KUKA KRL program: EPS_2_25694_BR06_A_20251117072402.src

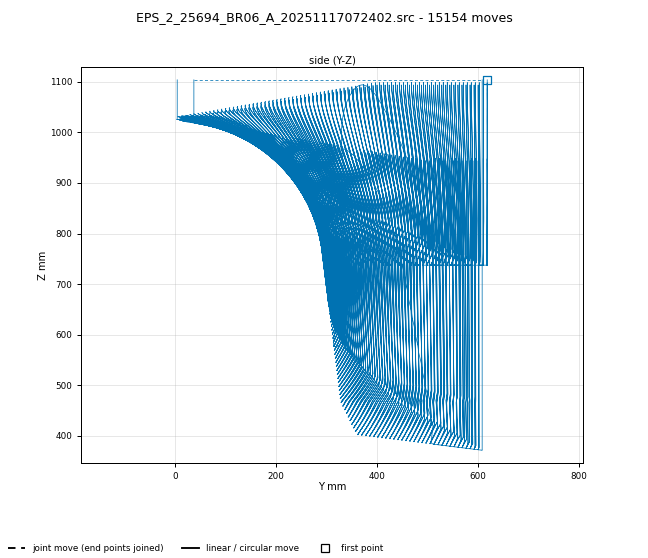
[picture p0: tool path of EPS_2_25694_BR06_A_20251117072402.src, 15154 of 15156 moves have a stored position in this frame; points joined in program order, loops and branches not executed]
&ACCESS RVP
&REL 4
&COMMENT QRS 19112012
&PARAM EDITMASK = *
DEF PART()
EXT BAS (BAS_COMMAND :IN,REAL :IN )
INT I
BAS (#INITMOV,0 )

;KUKA QRS Post kuka4.cps  Date:22-06-2017 !

File_ID=2908

QRS_PRE_INIT()

;Init var - Until changes are made in qrs_pre_init
Outlet_Square_prg=0
Inlet_1_Square_prg=0
Inlet_2_Square_prg=0
Inlet_3_Square_prg=0
Inlet_4_Square_prg=0
Inlet_5_Square_prg=0

Outlet_1={X 0.000, Y 400.000, Z 789.000, B 0.000, E1 0.000 }
Inlet_1={X 0.000, Y 466.000, Z 645.500, B 0.000, E1 180.000 }
Outlet_1_type=610
Inlet_1_type=457
;QRS#1=Sidecore dimensions
;QRS#2=600-24" Concrete
;QRS#3=450-18" Concrete
;QRS#4=
;QRS#5=
;QRS#6=
;QRS#7=
;QRS#8=
;QRS#9=S306-34L
;QRS#10=28A PSX-2
;QRS#11=
;QRS#12=
;QRS#13=
;QRS#14=
;QRS#15=
;QRS#16=1220x127x1448 4,75'
;QRS#17=EPS Height
;QRS#18=1094
;QRS#19=*
;QRS#20= UPDATED VERSION 22-06-2017
;QRS#21=*
Outlet_Square=0450
Inlet_1_Square=0250
Inlet_2_Square=0
Inlet_3_Square=0
Inlet_4_Square=0
Inlet_5_Square=0
Mill_Square=1
Outlet_Square_Prg=264
Inlet_1_Square_prg=274

QRS_INIT()

$ADVANCE=5

; T1
PTP {E1 171.024,E2 171.024}
PTP {X 0,Y 617.83,A -85,B 0,C 180,E1 171.024,E2 171.024,E3 0,E4 0,E5 0,E6 0}
QRS_SPEED_INIT()
LIN {X 0,Y 617.83,Z 1104,A -85,B 0,C 180,E1 171.024,E2 171.024,E3 0,E4 0,E5 0,E6 0} C_VEL
LIN {X 0,Y 617.83,Z 739.44,A -85,B 0,C 180,E1 171.024,E2 171.024} C_VEL
LIN {X 0,Y 617.865,Z 737.44,A -85,B 0,C 180,E1 171.21,E2 171.21} C_VEL
LIN {X 0,Y 618.044,Z 737.44,A -85,B 0,C 180,E1 171.886,E2 171.886} C_VEL
LIN {X 0,Y 618.018,Z 737.44,A -85,B 0,C 180,E1 176.532,E2 176.532} C_VEL
LIN {X 0,Y 618.01,Z 737.44,A -85,B 0,C 180,E1 181.155,E2 181.155} C_VEL
LIN {X 0,Y 617.998,Z 737.44,A -85,B 0,C 180,E1 185.786,E2 185.786} C_VEL
LIN {X 0,Y 618.001,Z 737.44,A -85,B 0,C 180,E1 190.456,E2 190.456} C_VEL
LIN {X 0,Y 617.923,Z 737.44,A -85,B 0,C 180,E1 195.199,E2 195.199} C_VEL
LIN {X 0,Y 617.894,Z 737.44,A -85,B 0,C 180,E1 200.05,E2 200.05} C_VEL
LIN {X 0,Y 617.438,Z 737.44,A -85,B 0,C 180,E1 202.548,E2 202.548} C_VEL
LIN {X 0,Y 617.919,Z 737.44,A -85,B 0,C 180,E1 205.056,E2 205.056} C_VEL
LIN {X 0,Y 617.398,Z 737.44,A -85,B 0,C 180,E1 207.66,E2 207.66} C_VEL
LIN {X 0,Y 617.828,Z 737.44,A -85,B 0,C 180,E1 210.281,E2 210.281} C_VEL
LIN {X 0,Y 617.3,Z 737.44,A -85,B 0,C 180,E1 213.028,E2 213.028} C_VEL
LIN {X 0,Y 617.772,Z 737.44,A -85,B 0,C 180,E1 215.801,E2 215.801} C_VEL
LIN {X 0,Y 617.531,Z 737.44,A -85,B 0,C 180,E1 218.094,E2 218.094} C_VEL
LIN {X 0,Y 617.504,Z 737.44,A -85,B 0,C 180,E1 218.725,E2 218.725} C_VEL
LIN {X 0,Y 617.717,Z 737.44,A -85,B 0,C 180,E1 221.737,E2 221.737} C_VEL
LIN {X 0,Y 617.832,Z 737.44,A -85,B 0,C 180,E1 225.095,E2 225.095} C_VEL
LIN {X 0,Y 617.441,Z 737.44,A -85,B 0,C 180,E1 228.309,E2 228.309} C_VEL
LIN {X 0,Y 617.823,Z 737.44,A -85,B 0,C 180,E1 231.298,E2 231.298} C_VEL
LIN {X 0,Y 617.894,Z 737.44,A -85,B 0,C 180,E1 235.778,E2 235.778} C_VEL
LIN {X 0,Y 617.659,Z 737.44,A -85,B 0,C 180,E1 236.368,E2 236.368} C_VEL
LIN {X 0,Y 616.896,Z 737.475,A -85,B 0,C 180,E1 236.468,E2 236.468} C_VEL
LIN {X 0,Y 617.501,Z 807.52,A -85,B 0,C 180,E1 237.463,E2 237.463} C_VEL
LIN {X 0,Y 617.519,Z 821.027,A -85,B 0,C 180,E1 237.687,E2 237.687} C_VEL
LIN {X 0,Y 617.637,Z 835.781,A -85,B 0,C 180,E1 238.01,E2 238.01} C_VEL
LIN {X 0,Y 617.583,Z 847.979,A -85,B 0,C 180,E1 238.328,E2 238.328} C_VEL
LIN {X 0,Y 617.775,Z 865.118,A -85,B 0,C 180,E1 238.871,E2 238.871} C_VEL
LIN {X 0,Y 617.661,Z 879.46,A -85,B 0,C 180,E1 239.394,E2 239.394} C_VEL
LIN {X 0,Y 617.795,Z 895.272,A -85,B 0,C 180,E1 240.077,E2 240.077} C_VEL
LIN {X 0,Y 617.796,Z 909.603,A -85,B 0,C 180,E1 240.772,E2 240.772} C_VEL
LIN {X 0,Y 617.753,Z 921.6,A -85,B 0,C 180,E1 241.411,E2 241.411} C_VEL
LIN {X 0,Y 617.843,Z 936.189,A -85,B 0,C 180,E1 242.286,E2 242.286} C_VEL
LIN {X 0,Y 617.842,Z 949.624,A -85,B 0,C 180,E1 243.174,E2 243.174} C_VEL
LIN {X 0,Y 617.833,Z 961.892,A -85,B 0,C 180,E1 244.06,E2 244.06} C_VEL
LIN {X 0,Y 617.824,Z 973.111,A -85,B 0,C 180,E1 244.94,E2 244.94} C_VEL
LIN {X 0,Y 617.855,Z 984.21,A -85,B 0,C 180,E1 245.886,E2 245.886} C_VEL
LIN {X 0,Y 617.904,Z 995.178,A -85,B 0,C 180,E1 246.901,E2 246.901} C_VEL
LIN {X 0,Y 617.833,Z 1005.53,A -85,B 0,C 180,E1 247.935,E2 247.935} C_VEL
LIN {X 0,Y 617.852,Z 1015.52,A -85,B 0,C 180,E1 249.023,E2 249.023} C_VEL
LIN {X 0,Y 617.958,Z 1024.894,A -85,B 0,C 180,E1 250.135,E2 250.135} C_VEL
LIN {X 0,Y 617.806,Z 1033.458,A -85,B 0,C 180,E1 251.226,E2 251.226} C_VEL
LIN {X 0,Y 617.799,Z 1041.796,A -85,B 0,C 180,E1 252.389,E2 252.389} C_VEL
LIN {X 0,Y 618,Z 1049.733,A -85,B 0,C 180,E1 253.612,E2 253.612} C_VEL
LIN {X 0,Y 617.809,Z 1056.882,A -85,B 0,C 180,E1 254.799,E2 254.799} C_VEL
LIN {X 0,Y 617.809,Z 1064.812,A -85,B 0,C 180,E1 256.29,E2 256.29} C_VEL
LIN {X 0,Y 617.96,Z 1070.477,A -85,B 0,C 180,E1 257.48,E2 257.48} C_VEL
LIN {X 0,Y 617.732,Z 1076.732,A -85,B 0,C 180,E1 258.951,E2 258.951} C_VEL
LIN {X 0,Y 617.808,Z 1081.629,A -85,B 0,C 180,E1 260.287,E2 260.287} C_VEL
LIN {X 0,Y 617.978,Z 1084.319,A -85,B 0,C 180,E1 261.142,E2 261.142} C_VEL
LIN {X 0,Y 617.858,Z 1086.559,A -85,B 0,C 180,E1 261.884,E2 261.884} C_VEL
LIN {X 0,Y 617.745,Z 1089.107,A -85,B 0,C 180,E1 262.815,E2 262.815} C_VEL
LIN {X 0,Y 617.831,Z 1092.206,A -85,B 0,C 180,E1 264.212,E2 264.212} C_VEL
LIN {X 0,Y 617.977,Z 1093.802,A -85,B 0,C 180,E1 265.142,E2 265.142} C_VEL
LIN {X 0,Y 617.8,Z 1095.279,A -85,B 0,C 180,E1 266.068,E2 266.068} C_VEL
LIN {X 0,Y 617.754,Z 1096.831,A -85,B 0,C 180,E1 267.456,E2 267.456} C_VEL
LIN {X 0,Y 617.996,Z 1097.642,A -85,B 0,C 180,E1 268.845,E2 268.845} C_VEL
LIN {X 0,Y 617.666,Z 1097.732,A -85,B 0,C 180,E1 271.156,E2 271.156} C_VEL
LIN {X 0,Y 617.779,Z 1097.15,A -85,B 0,C 180,E1 272.081,E2 272.081} C_VEL
LIN {X 0,Y 617.842,Z 1095.819,A -85,B 0,C 180,E1 273.469,E2 273.469} C_VEL
LIN {X 0,Y 617.71,Z 1093.872,A -85,B 0,C 180,E1 274.86,E2 274.86} C_VEL
LIN {X 0,Y 617.804,Z 1092.213,A -85,B 0,C 180,E1 275.788,E2 275.788} C_VEL
LIN {X 0,Y 617.987,Z 1090.125,A -85,B 0,C 180,E1 276.716,E2 276.716} C_VEL
LIN {X 0,Y 617.83,Z 1087.821,A -85,B 0,C 180,E1 277.65,E2 277.65} C_VEL
LIN {X 0,Y 617.78,Z 1084.463,A -85,B 0,C 180,E1 278.831,E2 278.831} C_VEL
LIN {X 0,Y 617.963,Z 1080.403,A -85,B 0,C 180,E1 280.049,E2 280.049} C_VEL
LIN {X 0,Y 617.795,Z 1075.563,A -85,B 0,C 180,E1 281.342,E2 281.342} C_VEL
LIN {X 0,Y 617.739,Z 1070.523,A -85,B 0,C 180,E1 282.524,E2 282.524} C_VEL
LIN {X 0,Y 617.973,Z 1063.299,A -85,B 0,C 180,E1 284.003,E2 284.003} C_VEL
LIN {X 0,Y 617.804,Z 1055.857,A -85,B 0,C 180,E1 285.375,E2 285.375} C_VEL
LIN {X 0,Y 617.794,Z 1048.024,A -85,B 0,C 180,E1 286.666,E2 286.666} C_VEL
LIN {X 0,Y 617.958,Z 1040.023,A -85,B 0,C 180,E1 287.859,E2 287.859} C_VEL
LIN {X 0,Y 617.819,Z 1031.946,A -85,B 0,C 180,E1 288.977,E2 288.977} C_VEL
LIN {X 0,Y 617.84,Z 1022.142,A -85,B 0,C 180,E1 290.206,E2 290.206} C_VEL
LIN {X 0,Y 617.954,Z 1012.763,A -85,B 0,C 180,E1 291.283,E2 291.283} C_VEL
LIN {X 0,Y 617.848,Z 1002.488,A -85,B 0,C 180,E1 292.376,E2 292.376} C_VEL
LIN {X 0,Y 617.845,Z 992.723,A -85,B 0,C 180,E1 293.335,E2 293.335} C_VEL
LIN {X 0,Y 617.862,Z 981.185,A -85,B 0,C 180,E1 294.376,E2 294.376} C_VEL
LIN {X 0,Y 617.853,Z 970.139,A -85,B 0,C 180,E1 295.298,E2 295.298} C_VEL
LIN {X 0,Y 617.84,Z 957.554,A -85,B 0,C 180,E1 296.261,E2 296.261} C_VEL
LIN {X 0,Y 617.827,Z 946.09,A -85,B 0,C 180,E1 297.07,E2 297.07} C_VEL
LIN {X 0,Y 617.852,Z 932.685,A -85,B 0,C 180,E1 297.929,E2 297.929} C_VEL
LIN {X 0,Y 617.813,Z 918.838,A -85,B 0,C 180,E1 298.735,E2 298.735} C_VEL
LIN {X 0,Y 617.728,Z 907.667,A -85,B 0,C 180,E1 299.334,E2 299.334} C_VEL
LIN {X 0,Y 617.8,Z 891.163,A -85,B 0,C 180,E1 300.105,E2 300.105} C_VEL
LIN {X 0,Y 617.676,Z 877.075,A -85,B 0,C 180,E1 300.695,E2 300.695} C_VEL
LIN {X 0,Y 617.673,Z 868.79,A -85,B 0,C 180,E1 301,E2 301} C_VEL
LIN {X 0,Y 617.767,Z 859.764,A -85,B 0,C 180,E1 301.301,E2 301.301} C_VEL
LIN {X 0,Y 617.783,Z 850.007,A -85,B 0,C 180,E1 301.607,E2 301.607} C_VEL
LIN {X 0,Y 617.56,Z 835.801,A -85,B 0,C 180,E1 301.994,E2 301.994} C_VEL
LIN {X 0,Y 617.673,Z 824.166,A -85,B 0,C 180,E1 302.238,E2 302.238} C_VEL
LIN {X 0,Y 617.731,Z 813.928,A -85,B 0,C 180,E1 302.42,E2 302.42} C_VEL
LIN {X 0,Y 617.65,Z 797.749,A -85,B 0,C 180,E1 302.666,E2 302.666} C_VEL
LIN {X 0,Y 616.962,Z 737.44,A -85,B 0,C 180,E1 303.538,E2 303.538} C_VEL
LIN {X 0,Y 617.672,Z 737.44,A -85,B 0,C 180,E1 303.632,E2 303.632} C_VEL
LIN {X 0,Y 617.852,Z 737.44,A -85,B 0,C 180,E1 304.322,E2 304.322} C_VEL
LIN {X 0,Y 617.822,Z 737.44,A -85,B 0,C 180,E1 308.702,E2 308.702} C_VEL
LIN {X 0,Y 617.438,Z 737.44,A -85,B 0,C 180,E1 311.761,E2 311.761} C_VEL
LIN {X 0,Y 617.832,Z 737.44,A -85,B 0,C 180,E1 314.905,E2 314.905} C_VEL
LIN {X 0,Y 617.712,Z 737.44,A -85,B 0,C 180,E1 318.281,E2 318.281} C_VEL
LIN {X 0,Y 617.499,Z 737.44,A -85,B 0,C 180,E1 321.274,E2 321.274} C_VEL
LIN {X 0,Y 617.532,Z 737.44,A -85,B 0,C 180,E1 321.905,E2 321.905} C_VEL
LIN {X 0,Y 617.768,Z 737.44,A -85,B 0,C 180,E1 324.199,E2 324.199} C_VEL
LIN {X 0,Y 617.292,Z 737.44,A -85,B 0,C 180,E1 326.972,E2 326.972} C_VEL
LIN {X 0,Y 617.823,Z 737.44,A -85,B 0,C 180,E1 329.719,E2 329.719} C_VEL
LIN {X 0,Y 617.394,Z 737.44,A -85,B 0,C 180,E1 332.34,E2 332.34} C_VEL
LIN {X 0,Y 617.916,Z 737.44,A -85,B 0,C 180,E1 334.944,E2 334.944} C_VEL
LIN {X 0,Y 617.434,Z 737.44,A -85,B 0,C 180,E1 337.451,E2 337.451} C_VEL
LIN {X 0,Y 617.912,Z 737.44,A -85,B 0,C 180,E1 339.95,E2 339.95} C_VEL
LIN {X 0,Y 618.008,Z 737.44,A -85,B 0,C 180,E1 343.638,E2 343.638} C_VEL
LIN {X 0,Y 617.998,Z 737.44,A -85,B 0,C 180,E1 349.544,E2 349.544} C_VEL
LIN {X 0,Y 618.008,Z 737.44,A -85,B 0,C 180,E1 354.214,E2 354.214} C_VEL
LIN {X 0,Y 618.008,Z 737.44,A -85,B 0,C 180,E1 358.845,E2 358.845} C_VEL
LIN {X 0,Y 618.014,Z 737.44,A -85,B 0,C 180,E1 363.468,E2 363.468} C_VEL
LIN {X 0,Y 618.049,Z 737.44,A -85,B 0,C 180,E1 368.114,E2 368.114} C_VEL
LIN {X 0,Y 617.956,Z 737.44,A -85,B 0,C 180,E1 372.816,E2 372.816} C_VEL
LIN {X 0,Y 617.925,Z 737.44,A -85,B 0,C 180,E1 377.608,E2 377.608} C_VEL
LIN {X 0,Y 617.741,Z 737.44,A -85,B 0,C 180,E1 378.539,E2 378.539} C_VEL
LIN {X 0,Y 617.936,Z 737.44,A -85,B 0,C 180,E1 382.529,E2 382.529} C_VEL
LIN {X 0,Y 617.421,Z 737.44,A -85,B 0,C 180,E1 385.077,E2 385.077} C_VEL
LIN {X 0,Y 617.843,Z 737.44,A -85,B 0,C 180,E1 387.638,E2 387.638} C_VEL
LIN {X 0,Y 617.351,Z 737.44,A -85,B 0,C 180,E1 390.307,E2 390.307} C_VEL
LIN {X 0,Y 617.847,Z 737.44,A -85,B 0,C 180,E1 392.995,E2 392.995} C_VEL
LIN {X 0,Y 617.706,Z 737.44,A -85,B 0,C 180,E1 394.196,E2 394.196} C_VEL
LIN {X 0,Y 617.767,Z 737.44,A -85,B 0,C 180,E1 398.706,E2 398.706} C_VEL
LIN {X 0,Y 617.422,Z 737.44,A -85,B 0,C 180,E1 401.762,E2 401.762} C_VEL
LIN {X 0,Y 617.834,Z 737.44,A -85,B 0,C 180,E1 404.905,E2 404.905} C_VEL
LIN {X 0,Y 617.74,Z 737.44,A -85,B 0,C 180,E1 408.278,E2 408.278} C_VEL
LIN {X 0,Y 617.526,Z 737.44,A -85,B 0,C 180,E1 411.276,E2 411.276} C_VEL
LIN {X 0,Y 617.553,Z 737.44,A -85,B 0,C 180,E1 411.903,E2 411.903} C_VEL
LIN {X 0,Y 617.798,Z 737.44,A -85,B 0,C 180,E1 414.201,E2 414.201} C_VEL
LIN {X 0,Y 617.326,Z 737.44,A -85,B 0,C 180,E1 416.974,E2 416.974} C_VEL
LIN {X 0,Y 617.834,Z 737.44,A -85,B 0,C 180,E1 419.719,E2 419.719} C_VEL
LIN {X 0,Y 618.015,Z 737.44,A -85,B 0,C 180,E1 425.143,E2 425.143} C_VEL
LIN {X 0,Y 617.953,Z 737.44,A -85,B 0,C 180,E1 425.36,E2 425.36} C_VEL
LIN {X 0,Y 616.403,Z 737.44,A -85,B 0,C 180,E1 425.601,E2 425.601} C_VEL
LIN {X 0,Y 617.555,Z 743.774,A -85,B 0,C 180,E1 425.777,E2 425.777} C_VEL
LIN {X 0,Y 617.78,Z 747.858,A -85,B 0,C 180,E1 425.88,E2 425.88} C_VEL
LIN {X 0,Y 617.88,Z 759.457,A -85,B 0,C 180,E1 426.181,E2 426.181} C_VEL
LIN {X 0,Y 617.842,Z 770.151,A -85,B 0,C 180,E1 426.503,E2 426.503} C_VEL
LIN {X 0,Y 617.91,Z 780.804,A -85,B 0,C 180,E1 426.879,E2 426.879} C_VEL
LIN {X 0,Y 617.941,Z 791.61,A -85,B 0,C 180,E1 427.313,E2 427.313} C_VEL
LIN {X 0,Y 617.864,Z 803.556,A -85,B 0,C 180,E1 427.858,E2 427.858} C_VEL
LIN {X 0,Y 617.94,Z 814.137,A -85,B 0,C 180,E1 428.406,E2 428.406} C_VEL
LIN {X 0,Y 617.955,Z 824.937,A -85,B 0,C 180,E1 429.026,E2 429.026} C_VEL
LIN {X 0,Y 617.944,Z 834.68,A -85,B 0,C 180,E1 429.643,E2 429.643} C_VEL
LIN {X 0,Y 617.95,Z 844.172,A -85,B 0,C 180,E1 430.304,E2 430.304} C_VEL
LIN {X 0,Y 617.931,Z 853.392,A -85,B 0,C 180,E1 431.007,E2 431.007} C_VEL
LIN {X 0,Y 617.961,Z 860.784,A -85,B 0,C 180,E1 431.618,E2 431.618} C_VEL
LIN {X 0,Y 617.973,Z 869.414,A -85,B 0,C 180,E1 432.394,E2 432.394} C_VEL
LIN {X 0,Y 617.911,Z 877.882,A -85,B 0,C 180,E1 433.225,E2 433.225} C_VEL
LIN {X 0,Y 617.922,Z 885.582,A -85,B 0,C 180,E1 434.052,E2 434.052} C_VEL
LIN {X 0,Y 617.992,Z 892.018,A -85,B 0,C 180,E1 434.803,E2 434.803} C_VEL
LIN {X 0,Y 617.915,Z 899.098,A -85,B 0,C 180,E1 435.697,E2 435.697} C_VEL
LIN {X 0,Y 617.864,Z 905.539,A -85,B 0,C 180,E1 436.589,E2 436.589} C_VEL
LIN {X 0,Y 617.934,Z 911.377,A -85,B 0,C 180,E1 437.48,E2 437.48} C_VEL
LIN {X 0,Y 617.935,Z 916.7,A -85,B 0,C 180,E1 438.366,E2 438.366} C_VEL
LIN {X 0,Y 617.82,Z 922.985,A -85,B 0,C 180,E1 439.541,E2 439.541} C_VEL
LIN {X 0,Y 617.872,Z 926.577,A -85,B 0,C 180,E1 440.284,E2 440.284} C_VEL
LIN {X 0,Y 617.957,Z 931.384,A -85,B 0,C 180,E1 441.413,E2 441.413} C_VEL
LIN {X 0,Y 617.813,Z 934.929,A -85,B 0,C 180,E1 442.35,E2 442.35} C_VEL
LIN {X 0,Y 617.786,Z 937.955,A -85,B 0,C 180,E1 443.281,E2 443.281} C_VEL
LIN {X 0,Y 617.98,Z 941.696,A -85,B 0,C 180,E1 444.678,E2 444.678} C_VEL
LIN {X 0,Y 617.786,Z 944.561,A -85,B 0,C 180,E1 446.067,E2 446.067} C_VEL
LIN {X 0,Y 617.783,Z 945.341,A -85,B 0,C 180,E1 446.531,E2 446.531} C_VEL
LIN {X 0,Y 617.939,Z 946.999,A -85,B 0,C 180,E1 447.92,E2 447.92} C_VEL
LIN {X 0,Y 617.892,Z 947.667,A -85,B 0,C 180,E1 448.844,E2 448.844} C_VEL
LIN {X 0,Y 617.796,Z 947.93,A -85,B 0,C 180,E1 449.769,E2 449.769} C_VEL
LIN {X 0,Y 617.897,Z 947.601,A -85,B 0,C 180,E1 451.156,E2 451.156} C_VEL
LIN {X 0,Y 617.872,Z 946.407,A -85,B 0,C 180,E1 452.543,E2 452.543} C_VEL
LIN {X 0,Y 617.786,Z 945.188,A -85,B 0,C 180,E1 453.469,E2 453.469} C_VEL
LIN {X 0,Y 617.788,Z 944.41,A -85,B 0,C 180,E1 453.933,E2 453.933} C_VEL
LIN {X 0,Y 617.98,Z 941.499,A -85,B 0,C 180,E1 455.322,E2 455.322} C_VEL
LIN {X 0,Y 617.846,Z 939.052,A -85,B 0,C 180,E1 456.253,E2 456.253} C_VEL
LIN {X 0,Y 617.872,Z 934.576,A -85,B 0,C 180,E1 457.649,E2 457.649} C_VEL
LIN {X 0,Y 617.982,Z 931.112,A -85,B 0,C 180,E1 458.565,E2 458.565} C_VEL
LIN {X 0,Y 617.843,Z 926.245,A -85,B 0,C 180,E1 459.696,E2 459.696} C_VEL
LIN {X 0,Y 617.859,Z 921.027,A -85,B 0,C 180,E1 460.752,E2 460.752} C_VEL
LIN {X 0,Y 617.982,Z 916.177,A -85,B 0,C 180,E1 461.633,E2 461.633} C_VEL
LIN {X 0,Y 617.909,Z 910.84,A -85,B 0,C 180,E1 462.521,E2 462.521} C_VEL
LIN {X 0,Y 617.877,Z 903.909,A -85,B 0,C 180,E1 463.559,E2 463.559} C_VEL
LIN {X 0,Y 617.982,Z 896.101,A -85,B 0,C 180,E1 464.599,E2 464.599} C_VEL
LIN {X 0,Y 617.951,Z 889.728,A -85,B 0,C 180,E1 465.384,E2 465.384} C_VEL
LIN {X 0,Y 617.903,Z 881.008,A -85,B 0,C 180,E1 466.358,E2 466.358} C_VEL
LIN {X 0,Y 617.954,Z 873.902,A -85,B 0,C 180,E1 467.085,E2 467.085} C_VEL
LIN {X 0,Y 617.962,Z 865.609,A -85,B 0,C 180,E1 467.865,E2 467.865} C_VEL
LIN {X 0,Y 617.941,Z 857.18,A -85,B 0,C 180,E1 468.594,E2 468.594} C_VEL
LIN {X 0,Y 617.945,Z 848.868,A -85,B 0,C 180,E1 469.256,E2 469.256} C_VEL
LIN {X 0,Y 617.954,Z 839.184,A -85,B 0,C 180,E1 469.96,E2 469.96} C_VEL
LIN {X 0,Y 617.95,Z 829.733,A -85,B 0,C 180,E1 470.588,E2 470.588} C_VEL
LIN {X 0,Y 617.916,Z 819.464,A -85,B 0,C 180,E1 471.207,E2 471.207} C_VEL
LIN {X 0,Y 617.939,Z 809.508,A -85,B 0,C 180,E1 471.75,E2 471.75} C_VEL
LIN {X 0,Y 617.952,Z 800.085,A -85,B 0,C 180,E1 472.216,E2 472.216} C_VEL
LIN {X 0,Y 617.928,Z 788.446,A -85,B 0,C 180,E1 472.728,E2 472.728} C_VEL
LIN {X 0,Y 617.799,Z 777.647,A -85,B 0,C 180,E1 473.151,E2 473.151} C_VEL
LIN {X 0,Y 617.942,Z 765.222,A -85,B 0,C 180,E1 473.558,E2 473.558} C_VEL
LIN {X 0,Y 617.928,Z 753.758,A -85,B 0,C 180,E1 473.88,E2 473.88} C_VEL
LIN {X 0,Y 617.77,Z 742.145,A -85,B 0,C 180,E1 474.156,E2 474.156} C_VEL
LIN {X 0,Y 617.503,Z 739.96,A -85,B 0,C 180,E1 474.209,E2 474.209} C_VEL
LIN {X 0,Y 616.484,Z 737.44,A -85,B 0,C 180,E1 474.307,E2 474.307} C_VEL
LIN {X 0,Y 617.908,Z 737.44,A -85,B 0,C 180,E1 474.586,E2 474.586} C_VEL
LIN {X 0,Y 617.983,Z 737.44,A -85,B 0,C 180,E1 475.053,E2 475.053} C_VEL
LIN {X 0,Y 617.957,Z 737.44,A -85,B 0,C 180,E1 477.633,E2 477.633} C_VEL
LIN {X 0,Y 617.388,Z 737.44,A -85,B 0,C 180,E1 480.305,E2 480.305} C_VEL
LIN {X 0,Y 617.865,Z 737.44,A -85,B 0,C 180,E1 482.994,E2 482.994} C_VEL
LIN {X 0,Y 617.727,Z 737.44,A -85,B 0,C 180,E1 484.199,E2 484.199} C_VEL
LIN {X 0,Y 617.751,Z 737.44,A -85,B 0,C 180,E1 488.707,E2 488.707} C_VEL
LIN {X 0,Y 617.415,Z 737.44,A -85,B 0,C 180,E1 491.762,E2 491.762} C_VEL
LIN {X 0,Y 617.839,Z 737.44,A -85,B 0,C 180,E1 494.904,E2 494.904} C_VEL
LIN {X 0,Y 617.74,Z 737.44,A -85,B 0,C 180,E1 498.278,E2 498.278} C_VEL
LIN {X 0,Y 617.515,Z 737.44,A -85,B 0,C 180,E1 501.276,E2 501.276} C_VEL
LIN {X 0,Y 617.771,Z 737.44,A -85,B 0,C 180,E1 504.199,E2 504.199} C_VEL
LIN {X 0,Y 617.303,Z 737.44,A -85,B 0,C 180,E1 506.972,E2 506.972} C_VEL
LIN {X 0,Y 617.829,Z 737.44,A -85,B 0,C 180,E1 509.719,E2 509.719} C_VEL
LIN {X 0,Y 617.384,Z 737.44,A -85,B 0,C 180,E1 512.339,E2 512.339} C_VEL
LIN {X 0,Y 617.894,Z 737.44,A -85,B 0,C 180,E1 514.943,E2 514.943} C_VEL
LIN {X 0,Y 617.442,Z 737.44,A -85,B 0,C 180,E1 517.452,E2 517.452} C_VEL
LIN {X 0,Y 617.947,Z 737.44,A -85,B 0,C 180,E1 519.951,E2 519.951} C_VEL
LIN {X 0,Y 617.728,Z 737.44,A -85,B 0,C 180,E1 522.387,E2 522.387} C_VEL
LIN {X 0,Y 617.807,Z 737.44,A -85,B 0,C 180,E1 524.799,E2 524.799} C_VEL
LIN {X 0,Y 617.962,Z 737.44,A -85,B 0,C 180,E1 527.184,E2 527.184} C_VEL
LIN {X 0,Y 617.865,Z 737.44,A -85,B 0,C 180,E1 531.21,E2 531.21} C_VEL
LIN {X 0,Y 615.332,Z 737.44,A -85,B 0,C 180,E1 532.406,E2 532.406} C_VEL
LIN {X 0,Y 609.728,Z 737.44,A -85,B 0,C 180,E1 534.193,E2 534.193} C_VEL
LIN {X 0,Y 609.637,Z 737.44,A -85,B 0,C 180,E1 534.4,E2 534.4} C_VEL
LIN {X 0,Y 609.619,Z 737.44,A -85,B 0,C 180,E1 538.581,E2 538.581} C_VEL
LIN {X 0,Y 609.649,Z 737.44,A -85,B 0,C 180,E1 542.85,E2 542.85} C_VEL
LIN {X 0,Y 609.697,Z 737.44,A -85,B 0,C 180,E1 547.135,E2 547.135} C_VEL
LIN {X 0,Y 609.756,Z 737.44,A -85,B 0,C 180,E1 551.46,E2 551.46} C_VEL
LIN {X 0,Y 609.758,Z 737.44,A -85,B 0,C 180,E1 555.853,E2 555.853} C_VEL
LIN {X 0,Y 609.908,Z 737.44,A -85,B 0,C 180,E1 560.338,E2 560.338} C_VEL
LIN {X 0,Y 610.002,Z 737.44,A -85,B 0,C 180,E1 564.958,E2 564.958} C_VEL
LIN {X 0,Y 609.747,Z 737.44,A -85,B 0,C 180,E1 569.777,E2 569.777} C_VEL
LIN {X 0,Y 609.682,Z 737.44,A -85,B 0,C 180,E1 576.584,E2 576.584} C_VEL
LIN {X 0,Y 609.73,Z 737.44,A -85,B 0,C 180,E1 582.101,E2 582.101} C_VEL
LIN {X 0,Y 609.502,Z 737.44,A -85,B 0,C 180,E1 587.881,E2 587.881} C_VEL
LIN {X 0,Y 609.562,Z 737.44,A -85,B 0,C 180,E1 592.636,E2 592.636} C_VEL
LIN {X 0,Y 609.894,Z 737.44,A -85,B 0,C 180,E1 596.018,E2 596.018} C_VEL
LIN {X 0,Y 610.896,Z 831.299,A -85,B 0,C 180,E1 597.514,E2 597.514} C_VEL
LIN {X 0,Y 610.871,Z 869.335,A -85,B 0,C 180,E1 598.636,E2 598.636} C_VEL
LIN {X 0,Y 610.74,Z 909.235,A -85,B 0,C 180,E1 600.38,E2 600.38} C_VEL
LIN {X 0,Y 610.584,Z 948.823,A -85,B 0,C 180,E1 602.771,E2 602.771} C_VEL
LIN {X 0,Y 610.358,Z 985.019,A -85,B 0,C 180,E1 605.646,E2 605.646} C_VEL
LIN {X 0,Y 610.19,Z 1016.967,A -85,B 0,C 180,E1 608.914,E2 608.914} C_VEL
LIN {X 0,Y 610.056,Z 1042.93,A -85,B 0,C 180,E1 612.301,E2 612.301} C_VEL
LIN {X 0,Y 610.008,Z 1064.721,A -85,B 0,C 180,E1 615.996,E2 615.996} C_VEL
LIN {X 0,Y 609.944,Z 1080.433,A -85,B 0,C 180,E1 619.633,E2 619.633} C_VEL
LIN {X 0,Y 609.927,Z 1090.985,A -85,B 0,C 180,E1 623.16,E2 623.16} C_VEL
LIN {X 0,Y 610.05,Z 1095.905,A -85,B 0,C 180,E1 625.73,E2 625.73} C_VEL
LIN {X 0,Y 610.113,Z 1098.656,A -85,B 0,C 180,E1 628.578,E2 628.578} C_VEL
LIN {X 0,Y 609.985,Z 1097.627,A -85,B 0,C 180,E1 632.845,E2 632.845} C_VEL
LIN {X 0,Y 610.093,Z 1090.333,A -85,B 0,C 180,E1 637.127,E2 637.127} C_VEL
LIN {X 0,Y 609.999,Z 1077.737,A -85,B 0,C 180,E1 641.09,E2 641.09} C_VEL
LIN {X 0,Y 610.061,Z 1060.705,A -85,B 0,C 180,E1 644.754,E2 644.754} C_VEL
LIN {X 0,Y 610.17,Z 1039.044,A -85,B 0,C 180,E1 648.256,E2 648.256} C_VEL
LIN {X 0,Y 610.294,Z 1011.943,A -85,B 0,C 180,E1 651.655,E2 651.655} C_VEL
LIN {X 0,Y 610.393,Z 979.466,A -85,B 0,C 180,E1 654.841,E2 654.841} C_VEL
LIN {X 0,Y 610.56,Z 944.376,A -85,B 0,C 180,E1 657.532,E2 657.532} C_VEL
LIN {X 0,Y 610.726,Z 905.417,A -85,B 0,C 180,E1 659.814,E2 659.814} C_VEL
LIN {X 0,Y 610.912,Z 865.209,A -85,B 0,C 180,E1 661.515,E2 661.515} C_VEL
LIN {X 0,Y 610.969,Z 824.561,A -85,B 0,C 180,E1 662.627,E2 662.627} C_VEL
LIN {X 0,Y 609.884,Z 737.44,A -85,B 0,C 180,E1 664.009,E2 664.009} C_VEL
LIN {X 0,Y 609.612,Z 737.44,A -85,B 0,C 180,E1 669.655,E2 669.655} C_VEL
LIN {X 0,Y 609.685,Z 737.44,A -85,B 0,C 180,E1 675.948,E2 675.948} C_VEL
LIN {X 0,Y 609.506,Z 737.44,A -85,B 0,C 180,E1 680.356,E2 680.356} C_VEL
LIN {X 0,Y 609.559,Z 737.44,A -85,B 0,C 180,E1 685.161,E2 685.161} C_VEL
LIN {X 0,Y 609.704,Z 737.44,A -85,B 0,C 180,E1 690.355,E2 690.355} C_VEL
LIN {X 0,Y 609.989,Z 737.44,A -85,B 0,C 180,E1 695.041,E2 695.041} C_VEL
LIN {X 0,Y 609.763,Z 737.44,A -85,B 0,C 180,E1 701.167,E2 701.167} C_VEL
LIN {X 0,Y 609.375,Z 737.44,A -85,B 0,C 180,E1 705.685,E2 705.685} C_VEL
LIN {X 0,Y 609.928,Z 737.44,A -85,B 0,C 180,E1 709.991,E2 709.991} C_VEL
LIN {X 0,Y 610.087,Z 737.44,A -85,B 0,C 180,E1 714.3,E2 714.3} C_VEL
LIN {X 0,Y 609.738,Z 737.44,A -85,B 0,C 180,E1 719.996,E2 719.996} C_VEL
LIN {X 0,Y 609.836,Z 737.44,A -85,B 0,C 180,E1 724.267,E2 724.267} C_VEL
LIN {X 0,Y 609.967,Z 737.44,A -85,B 0,C 180,E1 728.56,E2 728.56} C_VEL
LIN {X 0,Y 610.011,Z 737.44,A -85,B 0,C 180,E1 732.902,E2 732.902} C_VEL
LIN {X 0,Y 609.76,Z 737.44,A -85,B 0,C 180,E1 738.826,E2 738.826} C_VEL
LIN {X 0,Y 609.732,Z 737.44,A -85,B 0,C 180,E1 743.403,E2 743.403} C_VEL
LIN {X 0,Y 609.754,Z 737.44,A -85,B 0,C 180,E1 748.142,E2 748.142} C_VEL
LIN {X 0,Y 609.925,Z 737.44,A -85,B 0,C 180,E1 753.092,E2 753.092} C_VEL
LIN {X 0,Y 609.572,Z 737.44,A -85,B 0,C 180,E1 759.651,E2 759.651} C_VEL
LIN {X 0,Y 609.698,Z 737.44,A -85,B 0,C 180,E1 765.95,E2 765.95} C_VEL
LIN {X 0,Y 609.512,Z 737.44,A -85,B 0,C 180,E1 770.344,E2 770.344} C_VEL
LIN {X 0,Y 609.588,Z 737.44,A -85,B 0,C 180,E1 775.164,E2 775.164} C_VEL
LIN {X 0,Y 609.674,Z 737.44,A -85,B 0,C 180,E1 780.344,E2 780.344} C_VEL
LIN {X 0,Y 609.544,Z 737.44,A -85,B 0,C 180,E1 785.239,E2 785.239} C_VEL
LIN {X 0,Y 610.595,Z 780.27,A -85,B 0,C 180,E1 786.565,E2 786.565} C_VEL
LIN {X 0,Y 610.469,Z 814.705,A -85,B 0,C 180,E1 788.161,E2 788.161} C_VEL
LIN {X 0,Y 610.338,Z 846.661,A -85,B 0,C 180,E1 790.236,E2 790.236} C_VEL
LIN {X 0,Y 610.231,Z 876.67,A -85,B 0,C 180,E1 792.865,E2 792.865} C_VEL
LIN {X 0,Y 610.14,Z 901.637,A -85,B 0,C 180,E1 795.816,E2 795.816} C_VEL
LIN {X 0,Y 610.063,Z 921.017,A -85,B 0,C 180,E1 798.911,E2 798.911} C_VEL
LIN {X 0,Y 610.018,Z 936.047,A -85,B 0,C 180,E1 802.344,E2 802.344} C_VEL
LIN {X 0,Y 610.002,Z 945.047,A -85,B 0,C 180,E1 805.73,E2 805.73} C_VEL
LIN {X 0,Y 610.062,Z 948.539,A -85,B 0,C 180,E1 808.578,E2 808.578} C_VEL
LIN {X 0,Y 610.042,Z 948.475,A -85,B 0,C 180,E1 811.422,E2 811.422} C_VEL
LIN {X 0,Y 610.075,Z 943.354,A -85,B 0,C 180,E1 814.983,E2 814.983} C_VEL
LIN {X 0,Y 610.161,Z 932.33,A -85,B 0,C 180,E1 818.562,E2 818.562} C_VEL
LIN {X 0,Y 610.142,Z 915.442,A -85,B 0,C 180,E1 821.994,E2 821.994} C_VEL
LIN {X 0,Y 610.225,Z 895.319,A -85,B 0,C 180,E1 824.923,E2 824.923} C_VEL
LIN {X 0,Y 610.292,Z 870.045,A -85,B 0,C 180,E1 827.692,E2 827.692} C_VEL
LIN {X 0,Y 610.403,Z 839.47,A -85,B 0,C 180,E1 830.199,E2 830.199} C_VEL
LIN {X 0,Y 610.506,Z 807.616,A -85,B 0,C 180,E1 832.125,E2 832.125} C_VEL
LIN {X 0,Y 610.576,Z 773.34,A -85,B 0,C 180,E1 833.592,E2 833.592} C_VEL
LIN {X 0,Y 609.844,Z 741.091,A -85,B 0,C 180,E1 834.512,E2 834.512} C_VEL
LIN {X 0,Y 609.635,Z 737.44,A -85,B 0,C 180,E1 834.678,E2 834.678} C_VEL
LIN {X 0,Y 609.844,Z 737.44,A -85,B 0,C 180,E1 838.144,E2 838.144} C_VEL
LIN {X 0,Y 609.942,Z 737.44,A -85,B 0,C 180,E1 843.099,E2 843.099} C_VEL
LIN {X 0,Y 609.57,Z 737.44,A -85,B 0,C 180,E1 849.662,E2 849.662} C_VEL
LIN {X 0,Y 609.684,Z 737.44,A -85,B 0,C 180,E1 855.958,E2 855.958} C_VEL
LIN {X 0,Y 609.505,Z 737.44,A -85,B 0,C 180,E1 860.357,E2 860.357} C_VEL
LIN {X 0,Y 609.557,Z 737.44,A -85,B 0,C 180,E1 865.169,E2 865.169} C_VEL
LIN {X 0,Y 609.71,Z 737.44,A -85,B 0,C 180,E1 870.354,E2 870.354} C_VEL
LIN {X 0,Y 609.975,Z 737.44,A -85,B 0,C 180,E1 875.049,E2 875.049} C_VEL
LIN {X 0,Y 609.826,Z 737.44,A -85,B 0,C 180,E1 881.176,E2 881.176} C_VEL
LIN {X 0,Y 610.052,Z 737.44,A -85,B 0,C 180,E1 887.099,E2 887.099} C_VEL
LIN {X 0,Y 609.821,Z 737.44,A -85,B 0,C 180,E1 892.874,E2 892.874} C_VEL
LIN {X 0,Y 609.637,Z 737.44,A -85,B 0,C 180,E1 894.4,E2 894.4} C_VEL
LIN {X 0,Y 605.86,Z 737.44,A -85,B 0,C 180,E1 896.007,E2 896.007} C_VEL
LIN {X 0,Y 601.849,Z 737.44,A -85,B 0,C 180,E1 897.634,E2 897.634} C_VEL
LIN {X 0,Y 602.106,Z 737.44,A -85,B 0,C 180,E1 901.444,E2 901.444} C_VEL
LIN {X 0,Y 602.151,Z 737.44,A -85,B 0,C 180,E1 905.775,E2 905.775} C_VEL
LIN {X 0,Y 601.829,Z 737.44,A -85,B 0,C 180,E1 911.613,E2 911.613} C_VEL
LIN {X 0,Y 601.79,Z 737.44,A -85,B 0,C 180,E1 916.068,E2 916.068} C_VEL
LIN {X 0,Y 601.713,Z 737.44,A -85,B 0,C 180,E1 921.413,E2 921.413} C_VEL
LIN {X 0,Y 601.972,Z 737.44,A -85,B 0,C 180,E1 925.315,E2 925.315} C_VEL
LIN {X 0,Y 601.664,Z 737.44,A -85,B 0,C 180,E1 931.179,E2 931.179} C_VEL
LIN {X 0,Y 601.725,Z 737.44,A -85,B 0,C 180,E1 937.148,E2 937.148} C_VEL
LIN {X 0,Y 601.725,Z 737.44,A -85,B 0,C 180,E1 943.142,E2 943.142} C_VEL
LIN {X 0,Y 601.579,Z 737.44,A -85,B 0,C 180,E1 949.13,E2 949.13} C_VEL
LIN {X 0,Y 601.603,Z 737.44,A -85,B 0,C 180,E1 953.64,E2 953.64} C_VEL
LIN {X 0,Y 601.991,Z 737.44,A -85,B 0,C 180,E1 955.521,E2 955.521} C_VEL
LIN {X 0,Y 603.792,Z 744.834,A -85,B 0,C 180,E1 955.744,E2 955.744} C_VEL
LIN {X 0,Y 604.18,Z 830.014,A -85,B 0,C 180,E1 957.079,E2 957.079} C_VEL
LIN {X 0,Y 604.069,Z 867.838,A -85,B 0,C 180,E1 958.185,E2 958.185} C_VEL
LIN {X 0,Y 603.739,Z 908.692,A -85,B 0,C 180,E1 959.972,E2 959.972} C_VEL
LIN {X 0,Y 603.333,Z 947.771,A -85,B 0,C 180,E1 962.339,E2 962.339} C_VEL
LIN {X 0,Y 602.866,Z 985.013,A -85,B 0,C 180,E1 965.323,E2 965.323} C_VEL
LIN {X 0,Y 602.529,Z 1016.018,A -85,B 0,C 180,E1 968.519,E2 968.519} C_VEL
LIN {X 0,Y 602.264,Z 1042.932,A -85,B 0,C 180,E1 972.065,E2 972.065} C_VEL
LIN {X 0,Y 602.163,Z 1064.722,A -85,B 0,C 180,E1 975.81,E2 975.81} C_VEL
LIN {X 0,Y 602.064,Z 1080.737,A -85,B 0,C 180,E1 979.578,E2 979.578} C_VEL
LIN {X 0,Y 602.052,Z 1090.332,A -85,B 0,C 180,E1 982.777,E2 982.777} C_VEL
LIN {X 0,Y 602.172,Z 1095.905,A -85,B 0,C 180,E1 985.674,E2 985.674} C_VEL
LIN {X 0,Y 602.207,Z 1098.657,A -85,B 0,C 180,E1 988.559,E2 988.559} C_VEL
LIN {X 0,Y 602.081,Z 1097.627,A -85,B 0,C 180,E1 992.883,E2 992.883} C_VEL
LIN {X 0,Y 602.18,Z 1090.333,A -85,B 0,C 180,E1 997.222,E2 997.222} C_VEL
LIN {X 0,Y 602.129,Z 1077.488,A -85,B 0,C 180,E1 1001.305,E2 1001.305} C_VEL
LIN {X 0,Y 602.202,Z 1058.829,A -85,B 0,C 180,E1 1005.306,E2 1005.306} C_VEL
LIN {X 0,Y 602.339,Z 1035.021,A -85,B 0,C 180,E1 1009.072,E2 1009.072} C_VEL
LIN {X 0,Y 602.631,Z 1007.023,A -85,B 0,C 180,E1 1012.487,E2 1012.487} C_VEL
LIN {X 0,Y 602.98,Z 974.211,A -85,B 0,C 180,E1 1015.625,E2 1015.625} C_VEL
LIN {X 0,Y 603.418,Z 937.127,A -85,B 0,C 180,E1 1018.373,E2 1018.373} C_VEL
LIN {X 0,Y 603.807,Z 898.215,A -85,B 0,C 180,E1 1020.545,E2 1020.545} C_VEL
LIN {X 0,Y 604.137,Z 860.927,A -85,B 0,C 180,E1 1022.052,E2 1022.052} C_VEL
LIN {X 0,Y 604.372,Z 822.398,A -85,B 0,C 180,E1 1023.075,E2 1023.075} C_VEL
LIN {X 0,Y 603.314,Z 741.761,A -85,B 0,C 180,E1 1024.33,E2 1024.33} C_VEL
LIN {X 0,Y 602.006,Z 737.44,A -85,B 0,C 180,E1 1024.513,E2 1024.513} C_VEL
LIN {X 0,Y 601.78,Z 737.44,A -85,B 0,C 180,E1 1028.974,E2 1028.974} C_VEL
LIN {X 0,Y 601.692,Z 737.44,A -85,B 0,C 180,E1 1035.207,E2 1035.207} C_VEL
LIN {X 0,Y 601.696,Z 737.44,A -85,B 0,C 180,E1 1041.263,E2 1041.263} C_VEL
LIN {X 0,Y 601.492,Z 737.44,A -85,B 0,C 180,E1 1046.374,E2 1046.374} C_VEL
LIN {X 0,Y 601.616,Z 737.44,A -85,B 0,C 180,E1 1051.737,E2 1051.737} C_VEL
LIN {X 0,Y 601.719,Z 737.44,A -85,B 0,C 180,E1 1056.259,E2 1056.259} C_VEL
LIN {X 0,Y 601.903,Z 737.44,A -85,B 0,C 180,E1 1060.911,E2 1060.911} C_VEL
LIN {X 0,Y 601.526,Z 737.44,A -85,B 0,C 180,E1 1065.42,E2 1065.42} C_VEL
LIN {X 0,Y 601.984,Z 737.44,A -85,B 0,C 180,E1 1069.857,E2 1069.857} C_VEL
LIN {X 0,Y 602.175,Z 737.44,A -85,B 0,C 180,E1 1074.225,E2 1074.225} C_VEL
LIN {X 0,Y 601.837,Z 737.44,A -85,B 0,C 180,E1 1079.996,E2 1079.996} C_VEL
LIN {X 0,Y 601.949,Z 737.44,A -85,B 0,C 180,E1 1084.323,E2 1084.323} C_VEL
LIN {X 0,Y 602.023,Z 737.44,A -85,B 0,C 180,E1 1088.674,E2 1088.674} C_VEL
LIN {X 0,Y 602.035,Z 737.44,A -85,B 0,C 180,E1 1093.076,E2 1093.076} C_VEL
LIN {X 0,Y 601.818,Z 737.44,A -85,B 0,C 180,E1 1099.084,E2 1099.084} C_VEL
LIN {X 0,Y 601.756,Z 737.44,A -85,B 0,C 180,E1 1103.732,E2 1103.732} C_VEL
LIN {X 0,Y 601.737,Z 737.44,A -85,B 0,C 180,E1 1108.551,E2 1108.551} C_VEL
LIN {X 0,Y 601.811,Z 737.44,A -85,B 0,C 180,E1 1113.882,E2 1113.882} C_VEL
LIN {X 0,Y 601.729,Z 737.44,A -85,B 0,C 180,E1 1118.969,E2 1118.969} C_VEL
LIN {X 0,Y 601.7,Z 737.44,A -85,B 0,C 180,E1 1125.208,E2 1125.208} C_VEL
LIN {X 0,Y 601.694,Z 737.44,A -85,B 0,C 180,E1 1131.251,E2 1131.251} C_VEL
LIN {X 0,Y 601.519,Z 737.44,A -85,B 0,C 180,E1 1136.377,E2 1136.377} C_VEL
LIN {X 0,Y 601.532,Z 737.44,A -85,B 0,C 180,E1 1141.432,E2 1141.432} C_VEL
LIN {X 0,Y 602.035,Z 737.82,A -85,B 0,C 180,E1 1144.992,E2 1144.992} C_VEL
LIN {X 0,Y 603.332,Z 766.887,A -85,B 0,C 180,E1 1145.795,E2 1145.795} C_VEL
LIN {X 0,Y 603.098,Z 802.953,A -85,B 0,C 180,E1 1147.256,E2 1147.256} C_VEL
LIN {X 0,Y 602.859,Z 836.945,A -85,B 0,C 180,E1 1149.27,E2 1149.27} C_VEL
LIN {X 0,Y 602.62,Z 868.076,A -85,B 0,C 180,E1 1151.792,E2 1151.792} C_VEL
LIN {X 0,Y 602.473,Z 894.623,A -85,B 0,C 180,E1 1154.701,E2 1154.701} C_VEL
LIN {X 0,Y 602.28,Z 915.982,A -85,B 0,C 180,E1 1157.847,E2 1157.847} C_VEL
LIN {X 0,Y 602.235,Z 932.664,A -85,B 0,C 180,E1 1161.325,E2 1161.325} C_VEL
LIN {X 0,Y 602.189,Z 943.549,A -85,B 0,C 180,E1 1164.952,E2 1164.952} C_VEL
LIN {X 0,Y 602.158,Z 948.539,A -85,B 0,C 180,E1 1168.559,E2 1168.559} C_VEL
LIN {X 0,Y 602.139,Z 948.476,A -85,B 0,C 180,E1 1171.441,E2 1171.441} C_VEL
LIN {X 0,Y 602.19,Z 943.356,A -85,B 0,C 180,E1 1175.048,E2 1175.048} C_VEL
LIN {X 0,Y 602.261,Z 932.332,A -85,B 0,C 180,E1 1178.675,E2 1178.675} C_VEL
LIN {X 0,Y 602.312,Z 915.447,A -85,B 0,C 180,E1 1182.153,E2 1182.153} C_VEL
LIN {X 0,Y 602.444,Z 893.914,A -85,B 0,C 180,E1 1185.3,E2 1185.3} C_VEL
LIN {X 0,Y 602.628,Z 867.088,A -85,B 0,C 180,E1 1188.208,E2 1188.208} C_VEL
LIN {X 0,Y 602.869,Z 836.701,A -85,B 0,C 180,E1 1190.657,E2 1190.657} C_VEL
LIN {X 0,Y 603.163,Z 803.018,A -85,B 0,C 180,E1 1192.648,E2 1192.648} C_VEL
LIN {X 0,Y 603.409,Z 766.687,A -85,B 0,C 180,E1 1194.118,E2 1194.118} C_VEL
LIN {X 0,Y 602.681,Z 743.165,A -85,B 0,C 180,E1 1194.781,E2 1194.781} C_VEL
LIN {X 0,Y 602.17,Z 737.44,A -85,B 0,C 180,E1 1194.985,E2 1194.985} C_VEL
LIN {X 0,Y 601.573,Z 737.44,A -85,B 0,C 180,E1 1200.222,E2 1200.222} C_VEL
LIN {X 0,Y 601.823,Z 737.44,A -85,B 0,C 180,E1 1203.897,E2 1203.897} C_VEL
LIN {X 0,Y 601.722,Z 737.44,A -85,B 0,C 180,E1 1208.978,E2 1208.978} C_VEL
LIN {X 0,Y 601.692,Z 737.44,A -85,B 0,C 180,E1 1215.217,E2 1215.217} C_VEL
LIN {X 0,Y 601.636,Z 737.44,A -85,B 0,C 180,E1 1221.024,E2 1221.024} C_VEL
LIN {X 0,Y 601.506,Z 737.44,A -85,B 0,C 180,E1 1226.161,E2 1226.161} C_VEL
LIN {X 0,Y 601.611,Z 737.44,A -85,B 0,C 180,E1 1231.442,E2 1231.442} C_VEL
LIN {X 0,Y 601.728,Z 737.44,A -85,B 0,C 180,E1 1236.267,E2 1236.267} C_VEL
LIN {X 0,Y 601.95,Z 737.44,A -85,B 0,C 180,E1 1240.921,E2 1240.921} C_VEL
LIN {X 0,Y 602.107,Z 737.44,A -85,B 0,C 180,E1 1246.925,E2 1246.925} C_VEL
LIN {X 0,Y 601.923,Z 737.44,A -85,B 0,C 180,E1 1252.78,E2 1252.78} C_VEL
LIN {X 0,Y 601.849,Z 737.44,A -85,B 0,C 180,E1 1257.634,E2 1257.634} C_VEL
LIN {X 0,Y 597.786,Z 737.44,A -85,B 0,C 180,E1 1259.258,E2 1259.258} C_VEL
LIN {X 0,Y 594.059,Z 737.44,A -85,B 0,C 180,E1 1260.903,E2 1260.903} C_VEL
LIN {X 0,Y 594.083,Z 737.44,A -85,B 0,C 180,E1 1266.333,E2 1266.333} C_VEL
LIN {X 0,Y 593.892,Z 737.44,A -85,B 0,C 180,E1 1271.77,E2 1271.77} C_VEL
LIN {X 0,Y 593.845,Z 737.44,A -85,B 0,C 180,E1 1276.289,E2 1276.289} C_VEL
LIN {X 0,Y 593.93,Z 737.44,A -85,B 0,C 180,E1 1280.911,E2 1280.911} C_VEL
LIN {X 0,Y 593.951,Z 737.44,A -85,B 0,C 180,E1 1285.681,E2 1285.681} C_VEL
LIN {X 0,Y 593.786,Z 737.44,A -85,B 0,C 180,E1 1290.662,E2 1290.662} C_VEL
LIN {X 0,Y 593.795,Z 737.44,A -85,B 0,C 180,E1 1295.905,E2 1295.905} C_VEL
LIN {X 0,Y 593.744,Z 737.44,A -85,B 0,C 180,E1 1301.528,E2 1301.528} C_VEL
LIN {X 0,Y 593.679,Z 737.44,A -85,B 0,C 180,E1 1306.485,E2 1306.485} C_VEL
LIN {X 0,Y 593.78,Z 737.44,A -85,B 0,C 180,E1 1312.27,E2 1312.27} C_VEL
LIN {X 0,Y 593.922,Z 737.473,A -85,B 0,C 180,E1 1314.987,E2 1314.987} C_VEL
LIN {X 0,Y 597.258,Z 746.786,A -85,B 0,C 180,E1 1315.344,E2 1315.344} C_VEL
LIN {X 0,Y 597.533,Z 829.51,A -85,B 0,C 180,E1 1316.654,E2 1316.654} C_VEL
LIN {X 0,Y 597.252,Z 868.053,A -85,B 0,C 180,E1 1317.787,E2 1317.787} C_VEL
LIN {X 0,Y 596.741,Z 908.338,A -85,B 0,C 180,E1 1319.564,E2 1319.564} C_VEL
LIN {X 0,Y 596.078,Z 947.779,A -85,B 0,C 180,E1 1321.974,E2 1321.974} C_VEL
LIN {X 0,Y 595.446,Z 983.956,A -85,B 0,C 180,E1 1324.893,E2 1324.893} C_VEL
LIN {X 0,Y 594.916,Z 1016.019,A -85,B 0,C 180,E1 1328.23,E2 1328.23} C_VEL
LIN {X 0,Y 594.515,Z 1042.934,A -85,B 0,C 180,E1 1331.823,E2 1331.823} C_VEL
LIN {X 0,Y 594.319,Z 1063.96,A -85,B 0,C 180,E1 1335.469,E2 1335.469} C_VEL
LIN {X 0,Y 594.195,Z 1079.953,A -85,B 0,C 180,E1 1339.222,E2 1339.222} C_VEL
LIN {X 0,Y 594.162,Z 1090.332,A -85,B 0,C 180,E1 1342.68,E2 1342.68} C_VEL
LIN {X 0,Y 594.276,Z 1095.905,A -85,B 0,C 180,E1 1345.617,E2 1345.617} C_VEL
LIN {X 0,Y 594.3,Z 1098.657,A -85,B 0,C 180,E1 1348.54,E2 1348.54} C_VEL
LIN {X 0,Y 594.175,Z 1097.628,A -85,B 0,C 180,E1 1352.921,E2 1352.921} C_VEL
LIN {X 0,Y 594.294,Z 1090.333,A -85,B 0,C 180,E1 1357.318,E2 1357.318} C_VEL
LIN {X 0,Y 594.271,Z 1078.018,A -85,B 0,C 180,E1 1361.31,E2 1361.31} C_VEL
LIN {X 0,Y 594.397,Z 1060.802,A -85,B 0,C 180,E1 1365.134,E2 1365.134} C_VEL
LIN {X 0,Y 594.614,Z 1039.048,A -85,B 0,C 180,E1 1368.751,E2 1368.751} C_VEL
LIN {X 0,Y 594.999,Z 1011.625,A -85,B 0,C 180,E1 1372.276,E2 1372.276} C_VEL
LIN {X 0,Y 595.51,Z 979.73,A -85,B 0,C 180,E1 1375.483,E2 1375.483} C_VEL
LIN {X 0,Y 596.135,Z 943.82,A -85,B 0,C 180,E1 1378.296,E2 1378.296} C_VEL
LIN {X 0,Y 596.727,Z 905.846,A -85,B 0,C 180,E1 1380.566,E2 1380.566} C_VEL
LIN {X 0,Y 597.348,Z 865.28,A -85,B 0,C 180,E1 1382.314,E2 1382.314} C_VEL
LIN {X 0,Y 597.666,Z 825.786,A -85,B 0,C 180,E1 1383.42,E2 1383.42} C_VEL
LIN {X 0,Y 596.675,Z 744.205,A -85,B 0,C 180,E1 1384.732,E2 1384.732} C_VEL
LIN {X 0,Y 593.933,Z 737.44,A -85,B 0,C 180,E1 1385.08,E2 1385.08} C_VEL
LIN {X 0,Y 593.691,Z 737.44,A -85,B 0,C 180,E1 1390.089,E2 1390.089} C_VEL
LIN {X 0,Y 593.759,Z 737.44,A -85,B 0,C 180,E1 1395.557,E2 1395.557} C_VEL
LIN {X 0,Y 593.688,Z 737.44,A -85,B 0,C 180,E1 1400.391,E2 1400.391} C_VEL
LIN {X 0,Y 593.624,Z 737.44,A -85,B 0,C 180,E1 1405.867,E2 1405.867} C_VEL
LIN {X 0,Y 593.715,Z 737.44,A -85,B 0,C 180,E1 1411.018,E2 1411.018} C_VEL
LIN {X 0,Y 593.885,Z 737.44,A -85,B 0,C 180,E1 1415.926,E2 1415.926} C_VEL
LIN {X 0,Y 593.981,Z 737.44,A -85,B 0,C 180,E1 1420.647,E2 1420.647} C_VEL
LIN {X 0,Y 593.678,Z 737.44,A -85,B 0,C 180,E1 1425.223,E2 1425.223} C_VEL
LIN {X 0,Y 594.047,Z 737.44,A -85,B 0,C 180,E1 1429.72,E2 1429.72} C_VEL
LIN {X 0,Y 594.24,Z 737.44,A -85,B 0,C 180,E1 1434.147,E2 1434.147} C_VEL
LIN {X 0,Y 593.936,Z 737.44,A -85,B 0,C 180,E1 1439.996,E2 1439.996} C_VEL
LIN {X 0,Y 594.033,Z 737.44,A -85,B 0,C 180,E1 1444.381,E2 1444.381} C_VEL
LIN {X 0,Y 594.097,Z 737.44,A -85,B 0,C 180,E1 1448.791,E2 1448.791} C_VEL
LIN {X 0,Y 593.832,Z 737.44,A -85,B 0,C 180,E1 1454.346,E2 1454.346} C_VEL
LIN {X 0,Y 593.86,Z 737.44,A -85,B 0,C 180,E1 1459.39,E2 1459.39} C_VEL
LIN {X 0,Y 593.826,Z 737.44,A -85,B 0,C 180,E1 1464.068,E2 1464.068} C_VEL
LIN {X 0,Y 593.735,Z 737.44,A -85,B 0,C 180,E1 1468.972,E2 1468.972} C_VEL
LIN {X 0,Y 593.869,Z 737.44,A -85,B 0,C 180,E1 1474.108,E2 1474.108} C_VEL
LIN {X 0,Y 593.648,Z 737.44,A -85,B 0,C 180,E1 1480.085,E2 1480.085} C_VEL
LIN {X 0,Y 593.768,Z 737.44,A -85,B 0,C 180,E1 1485.547,E2 1485.547} C_VEL
LIN {X 0,Y 593.702,Z 737.44,A -85,B 0,C 180,E1 1490.393,E2 1490.393} C_VEL
LIN {X 0,Y 593.646,Z 737.44,A -85,B 0,C 180,E1 1495.87,E2 1495.87} C_VEL
LIN {X 0,Y 593.636,Z 737.44,A -85,B 0,C 180,E1 1501.016,E2 1501.016} C_VEL
LIN {X 0,Y 594.069,Z 737.539,A -85,B 0,C 180,E1 1504.628,E2 1504.628} C_VEL
LIN {X 0,Y 596.164,Z 757.647,A -85,B 0,C 180,E1 1505.203,E2 1505.203} C_VEL
LIN {X 0,Y 595.885,Z 793.964,A -85,B 0,C 180,E1 1506.536,E2 1506.536} C_VEL
LIN {X 0,Y 595.438,Z 828.145,A -85,B 0,C 180,E1 1508.402,E2 1508.402} C_VEL
LIN {X 0,Y 595.054,Z 859.697,A -85,B 0,C 180,E1 1510.782,E2 1510.782} C_VEL
LIN {X 0,Y 594.649,Z 887.317,A -85,B 0,C 180,E1 1513.595,E2 1513.595} C_VEL
LIN {X 0,Y 594.445,Z 910.424,A -85,B 0,C 180,E1 1516.749,E2 1516.749} C_VEL
LIN {X 0,Y 594.325,Z 928.122,A -85,B 0,C 180,E1 1520.099,E2 1520.099} C_VEL
LIN {X 0,Y 594.206,Z 940.141,A -85,B 0,C 180,E1 1523.485,E2 1523.485} C_VEL
LIN {X 0,Y 594.187,Z 947.22,A -85,B 0,C 180,E1 1527.079,E2 1527.079} C_VEL
LIN {X 0,Y 594.172,Z 948.996,A -85,B 0,C 180,E1 1530,E2 1530} C_VEL
LIN {X 0,Y 594.197,Z 946.094,A -85,B 0,C 180,E1 1533.652,E2 1533.652} C_VEL
LIN {X 0,Y 594.256,Z 937.466,A -85,B 0,C 180,E1 1537.319,E2 1537.319} C_VEL
LIN {X 0,Y 594.301,Z 924.681,A -85,B 0,C 180,E1 1540.555,E2 1540.555} C_VEL
LIN {X 0,Y 594.488,Z 906.427,A -85,B 0,C 180,E1 1543.779,E2 1543.779} C_VEL
LIN {X 0,Y 594.735,Z 881.544,A -85,B 0,C 180,E1 1546.974,E2 1546.974} C_VEL
LIN {X 0,Y 595.107,Z 854.218,A -85,B 0,C 180,E1 1549.591,E2 1549.591} C_VEL
LIN {X 0,Y 595.518,Z 821.39,A -85,B 0,C 180,E1 1551.936,E2 1551.936} C_VEL
LIN {X 0,Y 595.873,Z 786.616,A -85,B 0,C 180,E1 1553.697,E2 1553.697} C_VEL
LIN {X 0,Y 596.215,Z 750.117,A -85,B 0,C 180,E1 1554.902,E2 1554.902} C_VEL
LIN {X 0,Y 594.214,Z 737.44,A -85,B 0,C 180,E1 1555.29,E2 1555.29} C_VEL
LIN {X 0,Y 593.671,Z 737.44,A -85,B 0,C 180,E1 1560.667,E2 1560.667} C_VEL
LIN {X 0,Y 593.69,Z 737.44,A -85,B 0,C 180,E1 1565.323,E2 1565.323} C_VEL
LIN {X 0,Y 593.64,Z 737.44,A -85,B 0,C 180,E1 1570.095,E2 1570.095} C_VEL
LIN {X 0,Y 593.761,Z 737.44,A -85,B 0,C 180,E1 1575.558,E2 1575.558} C_VEL
LIN {X 0,Y 593.68,Z 737.44,A -85,B 0,C 180,E1 1580.4,E2 1580.4} C_VEL
LIN {X 0,Y 593.618,Z 737.44,A -85,B 0,C 180,E1 1585.876,E2 1585.876} C_VEL
LIN {X 0,Y 593.7,Z 737.44,A -85,B 0,C 180,E1 1591.026,E2 1591.026} C_VEL
LIN {X 0,Y 593.883,Z 737.44,A -85,B 0,C 180,E1 1595.934,E2 1595.934} C_VEL
LIN {X 0,Y 594.019,Z 737.44,A -85,B 0,C 180,E1 1600.656,E2 1600.656} C_VEL
LIN {X 0,Y 594.169,Z 737.44,A -85,B 0,C 180,E1 1606.748,E2 1606.748} C_VEL
LIN {X 0,Y 594.045,Z 737.44,A -85,B 0,C 180,E1 1612.683,E2 1612.683} C_VEL
LIN {X 0,Y 593.943,Z 737.44,A -85,B 0,C 180,E1 1617.618,E2 1617.618} C_VEL
LIN {X 0,Y 594.059,Z 737.44,A -85,B 0,C 180,E1 1620.903,E2 1620.903} C_VEL
LIN {X 0,Y 591.553,Z 737.44,A -85,B 0,C 180,E1 1622.147,E2 1622.147} C_VEL
LIN {X 0,Y 586.064,Z 737.44,A -85,B 0,C 180,E1 1624.008,E2 1624.008} C_VEL
LIN {X 0,Y 585.99,Z 737.44,A -85,B 0,C 180,E1 1624.223,E2 1624.223} C_VEL
LIN {X 0,Y 585.933,Z 737.44,A -85,B 0,C 180,E1 1628.922,E2 1628.922} C_VEL
LIN {X 0,Y 585.912,Z 737.44,A -85,B 0,C 180,E1 1633.451,E2 1633.451} C_VEL
LIN {X 0,Y 585.988,Z 737.44,A -85,B 0,C 180,E1 1639.628,E2 1639.628} C_VEL
LIN {X 0,Y 585.982,Z 737.44,A -85,B 0,C 180,E1 1646.056,E2 1646.056} C_VEL
LIN {X 0,Y 585.751,Z 737.44,A -85,B 0,C 180,E1 1651.466,E2 1651.466} C_VEL
LIN {X 0,Y 585.839,Z 737.44,A -85,B 0,C 180,E1 1656.761,E2 1656.761} C_VEL
LIN {X 0,Y 585.861,Z 737.44,A -85,B 0,C 180,E1 1662.214,E2 1662.214} C_VEL
LIN {X 0,Y 585.722,Z 737.44,A -85,B 0,C 180,E1 1667.774,E2 1667.774} C_VEL
LIN {X 0,Y 585.807,Z 737.44,A -85,B 0,C 180,E1 1673.243,E2 1673.243} C_VEL
LIN {X 0,Y 585.901,Z 737.44,A -85,B 0,C 180,E1 1674.417,E2 1674.417} C_VEL
LIN {X 0,Y 590.796,Z 749.203,A -85,B 0,C 180,E1 1674.945,E2 1674.945} C_VEL
LIN {X 0,Y 590.891,Z 829.509,A -85,B 0,C 180,E1 1676.229,E2 1676.229} C_VEL
LIN {X 0,Y 590.496,Z 868.051,A -85,B 0,C 180,E1 1677.373,E2 1677.373} C_VEL
LIN {X 0,Y 589.775,Z 908.335,A -85,B 0,C 180,E1 1679.165,E2 1679.165} C_VEL
LIN {X 0,Y 588.91,Z 946.803,A -85,B 0,C 180,E1 1681.531,E2 1681.531} C_VEL
LIN {X 0,Y 587.985,Z 984.547,A -85,B 0,C 180,E1 1684.609,E2 1684.609} C_VEL
LIN {X 0,Y 587.276,Z 1016.778,A -85,B 0,C 180,E1 1688.025,E2 1688.025} C_VEL
LIN {X 0,Y 586.753,Z 1042.936,A -85,B 0,C 180,E1 1691.574,E2 1691.574} C_VEL
LIN {X 0,Y 586.483,Z 1064.622,A -85,B 0,C 180,E1 1695.401,E2 1695.401} C_VEL
LIN {X 0,Y 586.339,Z 1080.505,A -85,B 0,C 180,E1 1699.23,E2 1699.23} C_VEL
LIN {X 0,Y 586.272,Z 1090.332,A -85,B 0,C 180,E1 1702.581,E2 1702.581} C_VEL
LIN {X 0,Y 586.38,Z 1095.905,A -85,B 0,C 180,E1 1705.557,E2 1705.557} C_VEL
LIN {X 0,Y 586.395,Z 1098.657,A -85,B 0,C 180,E1 1708.52,E2 1708.52} C_VEL
LIN {X 0,Y 586.278,Z 1097.628,A -85,B 0,C 180,E1 1712.96,E2 1712.96} C_VEL
LIN {X 0,Y 586.381,Z 1090.333,A -85,B 0,C 180,E1 1717.417,E2 1717.417} C_VEL
LIN {X 0,Y 586.378,Z 1078.002,A -85,B 0,C 180,E1 1721.469,E2 1721.469} C_VEL
LIN {X 0,Y 586.544,Z 1060.804,A -85,B 0,C 180,E1 1725.341,E2 1725.341} C_VEL
LIN {X 0,Y 586.864,Z 1039.05,A -85,B 0,C 180,E1 1729.008,E2 1729.008} C_VEL
LIN {X 0,Y 587.416,Z 1011.294,A -85,B 0,C 180,E1 1732.617,E2 1732.617} C_VEL
LIN {X 0,Y 588.111,Z 979.704,A -85,B 0,C 180,E1 1735.83,E2 1735.83} C_VEL
LIN {X 0,Y 588.942,Z 943.659,A -85,B 0,C 180,E1 1738.684,E2 1738.684} C_VEL
LIN {X 0,Y 589.778,Z 905.722,A -85,B 0,C 180,E1 1740.972,E2 1740.972} C_VEL
LIN {X 0,Y 590.598,Z 865.278,A -85,B 0,C 180,E1 1742.729,E2 1742.729} C_VEL
LIN {X 0,Y 591.052,Z 826.076,A -85,B 0,C 180,E1 1743.838,E2 1743.838} C_VEL
LIN {X 0,Y 590.184,Z 747.109,A -85,B 0,C 180,E1 1745.127,E2 1745.127} C_VEL
LIN {X 0,Y 585.905,Z 737.44,A -85,B 0,C 180,E1 1745.626,E2 1745.626} C_VEL
LIN {X 0,Y 585.714,Z 737.44,A -85,B 0,C 180,E1 1751.443,E2 1751.443} C_VEL
LIN {X 0,Y 585.886,Z 737.44,A -85,B 0,C 180,E1 1756.348,E2 1756.348} C_VEL
LIN {X 0,Y 585.812,Z 737.44,A -85,B 0,C 180,E1 1761.663,E2 1761.663} C_VEL
LIN {X 0,Y 585.688,Z 737.44,A -85,B 0,C 180,E1 1767.121,E2 1767.121} C_VEL
LIN {X 0,Y 585.767,Z 737.44,A -85,B 0,C 180,E1 1772.273,E2 1772.273} C_VEL
LIN {X 0,Y 585.842,Z 737.44,A -85,B 0,C 180,E1 1777.19,E2 1777.19} C_VEL
LIN {X 0,Y 586.055,Z 737.44,A -85,B 0,C 180,E1 1781.938,E2 1781.938} C_VEL
LIN {X 0,Y 585.805,Z 737.44,A -85,B 0,C 180,E1 1788.065,E2 1788.065} C_VEL
LIN {X 0,Y 586.316,Z 737.44,A -85,B 0,C 180,E1 1794.068,E2 1794.068} C_VEL
LIN {X 0,Y 586.047,Z 737.44,A -85,B 0,C 180,E1 1799.996,E2 1799.996} C_VEL
LIN {X 0,Y 586.124,Z 737.44,A -85,B 0,C 180,E1 1804.44,E2 1804.44} C_VEL
LIN {X 0,Y 586.157,Z 737.44,A -85,B 0,C 180,E1 1808.911,E2 1808.911} C_VEL
LIN {X 0,Y 586.126,Z 737.44,A -85,B 0,C 180,E1 1813.438,E2 1813.438} C_VEL
LIN {X 0,Y 585.956,Z 737.44,A -85,B 0,C 180,E1 1819.621,E2 1819.621} C_VEL
LIN {X 0,Y 585.862,Z 737.44,A -85,B 0,C 180,E1 1824.417,E2 1824.417} C_VEL
LIN {X 0,Y 585.766,Z 737.44,A -85,B 0,C 180,E1 1829.405,E2 1829.405} C_VEL
LIN {X 0,Y 585.885,Z 737.44,A -85,B 0,C 180,E1 1834.638,E2 1834.638} C_VEL
LIN {X 0,Y 585.753,Z 737.44,A -85,B 0,C 180,E1 1840.245,E2 1840.245} C_VEL
LIN {X 0,Y 585.887,Z 737.44,A -85,B 0,C 180,E1 1846.338,E2 1846.338} C_VEL
LIN {X 0,Y 585.807,Z 737.44,A -85,B 0,C 180,E1 1851.664,E2 1851.664} C_VEL
LIN {X 0,Y 585.711,Z 737.44,A -85,B 0,C 180,E1 1857.124,E2 1857.124} C_VEL
LIN {X 0,Y 585.663,Z 737.44,A -85,B 0,C 180,E1 1862.269,E2 1862.269} C_VEL
LIN {X 0,Y 586.039,Z 737.673,A -85,B 0,C 180,E1 1864.259,E2 1864.259} C_VEL
LIN {X 0,Y 588.95,Z 753.028,A -85,B 0,C 180,E1 1864.754,E2 1864.754} C_VEL
LIN {X 0,Y 588.607,Z 789.658,A -85,B 0,C 180,E1 1866.028,E2 1866.028} C_VEL
LIN {X 0,Y 588.061,Z 823.931,A -85,B 0,C 180,E1 1867.842,E2 1867.842} C_VEL
LIN {X 0,Y 587.471,Z 855.348,A -85,B 0,C 180,E1 1870.15,E2 1870.15} C_VEL
LIN {X 0,Y 586.983,Z 883.127,A -85,B 0,C 180,E1 1872.879,E2 1872.879} C_VEL
LIN {X 0,Y 586.671,Z 906.351,A -85,B 0,C 180,E1 1875.93,E2 1875.93} C_VEL
LIN {X 0,Y 586.438,Z 924.464,A -85,B 0,C 180,E1 1879.164,E2 1879.164} C_VEL
LIN {X 0,Y 586.318,Z 937.745,A -85,B 0,C 180,E1 1882.582,E2 1882.582} C_VEL
LIN {X 0,Y 586.33,Z 945.043,A -85,B 0,C 180,E1 1885.557,E2 1885.557} C_VEL
LIN {X 0,Y 586.351,Z 948.539,A -85,B 0,C 180,E1 1888.521,E2 1888.521} C_VEL
LIN {X 0,Y 586.334,Z 948.477,A -85,B 0,C 180,E1 1891.48,E2 1891.48} C_VEL
LIN {X 0,Y 586.428,Z 943.359,A -85,B 0,C 180,E1 1895.184,E2 1895.184} C_VEL
LIN {X 0,Y 586.468,Z 932.338,A -85,B 0,C 180,E1 1898.911,E2 1898.911} C_VEL
LIN {X 0,Y 586.592,Z 915.456,A -85,B 0,C 180,E1 1902.484,E2 1902.484} C_VEL
LIN {X 0,Y 586.901,Z 893.927,A -85,B 0,C 180,E1 1905.716,E2 1905.716} C_VEL
LIN {X 0,Y 587.301,Z 867.104,A -85,B 0,C 180,E1 1908.701,E2 1908.701} C_VEL
LIN {X 0,Y 587.806,Z 836.148,A -85,B 0,C 180,E1 1911.253,E2 1911.253} C_VEL
LIN {X 0,Y 588.465,Z 801.478,A -85,B 0,C 180,E1 1913.329,E2 1913.329} C_VEL
LIN {X 0,Y 588.956,Z 766.51,A -85,B 0,C 180,E1 1914.756,E2 1914.756} C_VEL
LIN {X 0,Y 588.101,Z 744.853,A -85,B 0,C 180,E1 1915.405,E2 1915.405} C_VEL
LIN {X 0,Y 586.251,Z 737.44,A -85,B 0,C 180,E1 1915.67,E2 1915.67} C_VEL
LIN {X 0,Y 585.791,Z 737.44,A -85,B 0,C 180,E1 1921.487,E2 1921.487} C_VEL
LIN {X 0,Y 585.891,Z 737.44,A -85,B 0,C 180,E1 1924.646,E2 1924.646} C_VEL
LIN {X 0,Y 585.745,Z 737.44,A -85,B 0,C 180,E1 1930.254,E2 1930.254} C_VEL
LIN {X 0,Y 585.885,Z 737.44,A -85,B 0,C 180,E1 1936.349,E2 1936.349} C_VEL
LIN {X 0,Y 585.777,Z 737.44,A -85,B 0,C 180,E1 1941.671,E2 1941.671} C_VEL
LIN {X 0,Y 585.681,Z 737.44,A -85,B 0,C 180,E1 1947.13,E2 1947.13} C_VEL
LIN {X 0,Y 585.753,Z 737.44,A -85,B 0,C 180,E1 1952.281,E2 1952.281} C_VEL
LIN {X 0,Y 585.851,Z 737.44,A -85,B 0,C 180,E1 1957.199,E2 1957.199} C_VEL
LIN {X 0,Y 586.039,Z 737.44,A -85,B 0,C 180,E1 1961.946,E2 1961.946} C_VEL
LIN {X 0,Y 586.247,Z 737.44,A -85,B 0,C 180,E1 1966.565,E2 1966.565} C_VEL
LIN {X 0,Y 586.14,Z 737.44,A -85,B 0,C 180,E1 1972.584,E2 1972.584} C_VEL
LIN {X 0,Y 586.19,Z 737.44,A -85,B 0,C 180,E1 1977.043,E2 1977.043} C_VEL
LIN {X 0,Y 586.292,Z 737.44,A -85,B 0,C 180,E1 1981.483,E2 1981.483} C_VEL
LIN {X 0,Y 585.99,Z 737.44,A -85,B 0,C 180,E1 1984.223,E2 1984.223} C_VEL
LIN {X 0,Y 583.567,Z 737.44,A -85,B 0,C 180,E1 1985.487,E2 1985.487} C_VEL
LIN {X 0,Y 578.052,Z 737.44,A -85,B 0,C 180,E1 1987.596,E2 1987.596} C_VEL
LIN {X 0,Y 578.057,Z 737.44,A -85,B 0,C 180,E1 1992.098,E2 1992.098} C_VEL
LIN {X 0,Y 577.982,Z 737.44,A -85,B 0,C 180,E1 1996.749,E2 1996.749} C_VEL
LIN {X 0,Y 578.026,Z 737.44,A -85,B 0,C 180,E1 2001.514,E2 2001.514} C_VEL
LIN {X 0,Y 577.914,Z 737.44,A -85,B 0,C 180,E1 2007.037,E2 2007.037} C_VEL
LIN {X 0,Y 577.798,Z 737.44,A -85,B 0,C 180,E1 2013.019,E2 2013.019} C_VEL
LIN {X 0,Y 577.888,Z 737.44,A -85,B 0,C 180,E1 2018.961,E2 2018.961} C_VEL
LIN {X 0,Y 577.901,Z 737.44,A -85,B 0,C 180,E1 2025.02,E2 2025.02} C_VEL
LIN {X 0,Y 577.919,Z 737.44,A -85,B 0,C 180,E1 2031.043,E2 2031.043} C_VEL
LIN {X 0,Y 577.93,Z 737.44,A -85,B 0,C 180,E1 2033.851,E2 2033.851} C_VEL
LIN {X 0,Y 584.245,Z 751.175,A -85,B 0,C 180,E1 2034.522,E2 2034.522} C_VEL
LIN {X 0,Y 584.316,Z 831.785,A -85,B 0,C 180,E1 2035.849,E2 2035.849} C_VEL
LIN {X 0,Y 583.712,Z 870.687,A -85,B 0,C 180,E1 2037.05,E2 2037.05} C_VEL
LIN {X 0,Y 582.797,Z 909.874,A -85,B 0,C 180,E1 2038.843,E2 2038.843} C_VEL
LIN {X 0,Y 581.683,Z 947.944,A -85,B 0,C 180,E1 2041.23,E2 2041.23} C_VEL
LIN {X 0,Y 580.568,Z 984.772,A -85,B 0,C 180,E1 2044.284,E2 2044.284} C_VEL
LIN {X 0,Y 579.657,Z 1015.915,A -85,B 0,C 180,E1 2047.613,E2 2047.613} C_VEL
LIN {X 0,Y 578.99,Z 1043.052,A -85,B 0,C 180,E1 2051.336,E2 2051.336} C_VEL
LIN {X 0,Y 578.66,Z 1064.755,A -85,B 0,C 180,E1 2055.227,E2 2055.227} C_VEL
LIN {X 0,Y 578.462,Z 1080.506,A -85,B 0,C 180,E1 2059.081,E2 2059.081} C_VEL
LIN {X 0,Y 578.398,Z 1090.332,A -85,B 0,C 180,E1 2062.48,E2 2062.48} C_VEL
LIN {X 0,Y 578.484,Z 1095.905,A -85,B 0,C 180,E1 2065.497,E2 2065.497} C_VEL
LIN {X 0,Y 578.489,Z 1098.657,A -85,B 0,C 180,E1 2068.5,E2 2068.5} C_VEL
LIN {X 0,Y 578.372,Z 1097.628,A -85,B 0,C 180,E1 2073.001,E2 2073.001} C_VEL
LIN {X 0,Y 578.512,Z 1091.917,A -85,B 0,C 180,E1 2076.763,E2 2076.763} C_VEL
LIN {X 0,Y 578.562,Z 1081.78,A -85,B 0,C 180,E1 2080.555,E2 2080.555} C_VEL
LIN {X 0,Y 578.743,Z 1064.617,A -85,B 0,C 180,E1 2084.799,E2 2084.799} C_VEL
LIN {X 0,Y 579.091,Z 1041.915,A -85,B 0,C 180,E1 2088.845,E2 2088.845} C_VEL
LIN {X 0,Y 579.79,Z 1013.997,A -85,B 0,C 180,E1 2092.619,E2 2092.619} C_VEL
LIN {X 0,Y 580.681,Z 981.083,A -85,B 0,C 180,E1 2096.06,E2 2096.06} C_VEL
LIN {X 0,Y 581.736,Z 945.464,A -85,B 0,C 180,E1 2098.947,E2 2098.947} C_VEL
LIN {X 0,Y 582.865,Z 906.067,A -85,B 0,C 180,E1 2101.364,E2 2101.364} C_VEL
LIN {X 0,Y 583.856,Z 865.999,A -85,B 0,C 180,E1 2103.126,E2 2103.126} C_VEL
LIN {X 0,Y 584.495,Z 825.695,A -85,B 0,C 180,E1 2104.278,E2 2104.278} C_VEL
LIN {X 0,Y 583.796,Z 750.336,A -85,B 0,C 180,E1 2105.522,E2 2105.522} C_VEL
LIN {X 0,Y 577.937,Z 737.44,A -85,B 0,C 180,E1 2106.184,E2 2106.184} C_VEL
LIN {X 0,Y 577.83,Z 737.44,A -85,B 0,C 180,E1 2110.922,E2 2110.922} C_VEL
LIN {X 0,Y 577.928,Z 737.44,A -85,B 0,C 180,E1 2117.068,E2 2117.068} C_VEL
LIN {X 0,Y 577.92,Z 737.44,A -85,B 0,C 180,E1 2122.947,E2 2122.947} C_VEL
LIN {X 0,Y 577.852,Z 737.44,A -85,B 0,C 180,E1 2128.397,E2 2128.397} C_VEL
LIN {X 0,Y 577.983,Z 737.44,A -85,B 0,C 180,E1 2133.555,E2 2133.555} C_VEL
LIN {X 0,Y 578.021,Z 737.44,A -85,B 0,C 180,E1 2138.486,E2 2138.486} C_VEL
LIN {X 0,Y 578.18,Z 737.44,A -85,B 0,C 180,E1 2143.257,E2 2143.257} C_VEL
LIN {X 0,Y 578.169,Z 737.44,A -85,B 0,C 180,E1 2149.435,E2 2149.435} C_VEL
LIN {X 0,Y 578.417,Z 737.44,A -85,B 0,C 180,E1 2154.063,E2 2154.063} C_VEL
LIN {X 0,Y 578.146,Z 737.44,A -85,B 0,C 180,E1 2159.996,E2 2159.996} C_VEL
LIN {X 0,Y 578.209,Z 737.44,A -85,B 0,C 180,E1 2164.501,E2 2164.501} C_VEL
LIN {X 0,Y 578.221,Z 737.44,A -85,B 0,C 180,E1 2169.034,E2 2169.034} C_VEL
LIN {X 0,Y 578.024,Z 737.44,A -85,B 0,C 180,E1 2174.276,E2 2174.276} C_VEL
LIN {X 0,Y 578.027,Z 737.44,A -85,B 0,C 180,E1 2179.902,E2 2179.902} C_VEL
LIN {X 0,Y 577.949,Z 737.44,A -85,B 0,C 180,E1 2184.773,E2 2184.773} C_VEL
LIN {X 0,Y 577.802,Z 737.44,A -85,B 0,C 180,E1 2190.153,E2 2190.153} C_VEL
LIN {X 0,Y 577.856,Z 737.44,A -85,B 0,C 180,E1 2195.19,E2 2195.19} C_VEL
LIN {X 0,Y 577.794,Z 737.44,A -85,B 0,C 180,E1 2200.916,E2 2200.916} C_VEL
LIN {X 0,Y 577.947,Z 737.44,A -85,B 0,C 180,E1 2207.071,E2 2207.071} C_VEL
LIN {X 0,Y 577.921,Z 737.44,A -85,B 0,C 180,E1 2212.948,E2 2212.948} C_VEL
LIN {X 0,Y 577.864,Z 737.44,A -85,B 0,C 180,E1 2218.4,E2 2218.4} C_VEL
LIN {X 0,Y 578.038,Z 737.584,A -85,B 0,C 180,E1 2223.875,E2 2223.875} C_VEL
LIN {X 0,Y 581.726,Z 752.639,A -85,B 0,C 180,E1 2224.408,E2 2224.408} C_VEL
LIN {X 0,Y 581.339,Z 789.307,A -85,B 0,C 180,E1 2225.695,E2 2225.695} C_VEL
LIN {X 0,Y 580.644,Z 823.517,A -85,B 0,C 180,E1 2227.518,E2 2227.518} C_VEL
LIN {X 0,Y 579.868,Z 855.898,A -85,B 0,C 180,E1 2229.927,E2 2229.927} C_VEL
LIN {X 0,Y 579.27,Z 883.453,A -85,B 0,C 180,E1 2232.681,E2 2232.681} C_VEL
LIN {X 0,Y 578.853,Z 907.116,A -85,B 0,C 180,E1 2235.859,E2 2235.859} C_VEL
LIN {X 0,Y 578.621,Z 924.461,A -85,B 0,C 180,E1 2239.016,E2 2239.016} C_VEL
LIN {X 0,Y 578.454,Z 937.743,A -85,B 0,C 180,E1 2242.481,E2 2242.481} C_VEL
LIN {X 0,Y 578.432,Z 946.24,A -85,B 0,C 180,E1 2246.248,E2 2246.248} C_VEL
LIN {X 0,Y 578.373,Z 948.997,A -85,B 0,C 180,E1 2250,E2 2250} C_VEL
LIN {X 0,Y 578.434,Z 946.097,A -85,B 0,C 180,E1 2253.752,E2 2253.752} C_VEL
LIN {X 0,Y 578.49,Z 937.47,A -85,B 0,C 180,E1 2257.519,E2 2257.519} C_VEL
LIN {X 0,Y 578.642,Z 924.041,A -85,B 0,C 180,E1 2260.986,E2 2260.986} C_VEL
LIN {X 0,Y 578.945,Z 903.978,A -85,B 0,C 180,E1 2264.533,E2 2264.533} C_VEL
LIN {X 0,Y 579.385,Z 879.37,A -85,B 0,C 180,E1 2267.682,E2 2267.682} C_VEL
LIN {X 0,Y 580.034,Z 850.643,A -85,B 0,C 180,E1 2270.432,E2 2270.432} C_VEL
LIN {X 0,Y 580.728,Z 818.529,A -85,B 0,C 180,E1 2272.699,E2 2272.699} C_VEL
LIN {X 0,Y 581.284,Z 784.595,A -85,B 0,C 180,E1 2274.417,E2 2274.417} C_VEL
LIN {X 0,Y 581.317,Z 748.657,A -85,B 0,C 180,E1 2275.625,E2 2275.625} C_VEL
LIN {X 0,Y 578.31,Z 737.44,A -85,B 0,C 180,E1 2276.068,E2 2276.068} C_VEL
LIN {X 0,Y 578.041,Z 737.44,A -85,B 0,C 180,E1 2283.071,E2 2283.071} C_VEL
LIN {X 0,Y 577.838,Z 737.44,A -85,B 0,C 180,E1 2288.963,E2 2288.963} C_VEL
LIN {X 0,Y 577.911,Z 737.44,A -85,B 0,C 180,E1 2295.019,E2 2295.019} C_VEL
LIN {X 0,Y 577.86,Z 737.44,A -85,B 0,C 180,E1 2301.047,E2 2301.047} C_VEL
LIN {X 0,Y 577.788,Z 737.44,A -85,B 0,C 180,E1 2306.982,E2 2306.982} C_VEL
LIN {X 0,Y 577.858,Z 737.44,A -85,B 0,C 180,E1 2311.869,E2 2311.869} C_VEL
LIN {X 0,Y 577.935,Z 737.44,A -85,B 0,C 180,E1 2316.868,E2 2316.868} C_VEL
LIN {X 0,Y 578.121,Z 737.44,A -85,B 0,C 180,E1 2321.69,E2 2321.69} C_VEL
LIN {X 0,Y 578.308,Z 737.44,A -85,B 0,C 180,E1 2326.377,E2 2326.377} C_VEL
LIN {X 0,Y 578.232,Z 737.44,A -85,B 0,C 180,E1 2332.482,E2 2332.482} C_VEL
LIN {X 0,Y 578.283,Z 737.44,A -85,B 0,C 180,E1 2337.003,E2 2337.003} C_VEL
LIN {X 0,Y 578.382,Z 737.44,A -85,B 0,C 180,E1 2341.504,E2 2341.504} C_VEL
LIN {X 0,Y 578.376,Z 737.44,A -85,B 0,C 180,E1 2346.014,E2 2346.014} C_VEL
LIN {X 0,Y 578.052,Z 737.44,A -85,B 0,C 180,E1 2347.596,E2 2347.596} C_VEL
LIN {X 0,Y 574.162,Z 737.44,A -85,B 0,C 180,E1 2349.288,E2 2349.288} C_VEL
LIN {X 0,Y 570.222,Z 737.44,A -85,B 0,C 180,E1 2351.003,E2 2351.003} C_VEL
LIN {X 0,Y 570.036,Z 737.44,A -85,B 0,C 180,E1 2357.031,E2 2357.031} C_VEL
LIN {X 0,Y 570.096,Z 737.44,A -85,B 0,C 180,E1 2361.829,E2 2361.829} C_VEL
LIN {X 0,Y 570.045,Z 737.44,A -85,B 0,C 180,E1 2366.842,E2 2366.842} C_VEL
LIN {X 0,Y 569.896,Z 737.44,A -85,B 0,C 180,E1 2372.097,E2 2372.097} C_VEL
LIN {X 0,Y 569.982,Z 737.44,A -85,B 0,C 180,E1 2377.658,E2 2377.658} C_VEL
LIN {X 0,Y 569.934,Z 737.44,A -85,B 0,C 180,E1 2383.684,E2 2383.684} C_VEL
LIN {X 0,Y 569.857,Z 737.44,A -85,B 0,C 180,E1 2388.379,E2 2388.379} C_VEL
LIN {X 0,Y 569.993,Z 737.44,A -85,B 0,C 180,E1 2393.277,E2 2393.277} C_VEL
LIN {X 0,Y 576.276,Z 751.195,A -85,B 0,C 180,E1 2393.956,E2 2393.956} C_VEL
LIN {X 0,Y 577.915,Z 755.058,A -85,B 0,C 180,E1 2394.132,E2 2394.132} C_VEL
LIN {X 0,Y 577.756,Z 831.642,A -85,B 0,C 180,E1 2395.403,E2 2395.403} C_VEL
LIN {X 0,Y 576.991,Z 870.752,A -85,B 0,C 180,E1 2396.619,E2 2396.619} C_VEL
LIN {X 0,Y 575.896,Z 909.23,A -85,B 0,C 180,E1 2398.39,E2 2398.39} C_VEL
LIN {X 0,Y 574.538,Z 947.585,A -85,B 0,C 180,E1 2400.81,E2 2400.81} C_VEL
LIN {X 0,Y 573.168,Z 984.576,A -85,B 0,C 180,E1 2403.908,E2 2403.908} C_VEL
LIN {X 0,Y 572.067,Z 1016.144,A -85,B 0,C 180,E1 2407.328,E2 2407.328} C_VEL
LIN {X 0,Y 571.272,Z 1043.25,A -85,B 0,C 180,E1 2411.107,E2 2411.107} C_VEL
LIN {X 0,Y 570.823,Z 1064.44,A -85,B 0,C 180,E1 2414.954,E2 2414.954} C_VEL
LIN {X 0,Y 570.603,Z 1080.846,A -85,B 0,C 180,E1 2419.027,E2 2419.027} C_VEL
LIN {X 0,Y 570.514,Z 1090.332,A -85,B 0,C 180,E1 2422.375,E2 2422.375} C_VEL
LIN {X 0,Y 570.613,Z 1095.905,A -85,B 0,C 180,E1 2425.434,E2 2425.434} C_VEL
LIN {X 0,Y 570.59,Z 1098.657,A -85,B 0,C 180,E1 2428.479,E2 2428.479} C_VEL
LIN {X 0,Y 570.466,Z 1097.628,A -85,B 0,C 180,E1 2433.043,E2 2433.043} C_VEL
LIN {X 0,Y 570.605,Z 1091.918,A -85,B 0,C 180,E1 2436.857,E2 2436.857} C_VEL
LIN {X 0,Y 570.657,Z 1080.745,A -85,B 0,C 180,E1 2441.002,E2 2441.002} C_VEL
LIN {X 0,Y 570.925,Z 1064.317,A -85,B 0,C 180,E1 2445.067,E2 2445.067} C_VEL
LIN {X 0,Y 571.346,Z 1041.124,A -85,B 0,C 180,E1 2449.231,E2 2449.231} C_VEL
LIN {X 0,Y 572.194,Z 1013.181,A -85,B 0,C 180,E1 2453.032,E2 2453.032} C_VEL
LIN {X 0,Y 573.319,Z 980.377,A -85,B 0,C 180,E1 2456.485,E2 2456.485} C_VEL
LIN {X 0,Y 574.64,Z 944.317,A -85,B 0,C 180,E1 2459.421,E2 2459.421} C_VEL
LIN {X 0,Y 575.982,Z 905.982,A -85,B 0,C 180,E1 2461.786,E2 2461.786} C_VEL
LIN {X 0,Y 577.149,Z 865.997,A -85,B 0,C 180,E1 2463.562,E2 2463.562} C_VEL
LIN {X 0,Y 577.92,Z 827.292,A -85,B 0,C 180,E1 2464.687,E2 2464.687} C_VEL
LIN {X 0,Y 577.497,Z 753.333,A -85,B 0,C 180,E1 2465.924,E2 2465.924} C_VEL
LIN {X 0,Y 569.995,Z 737.44,A -85,B 0,C 180,E1 2466.811,E2 2466.811} C_VEL
LIN {X 0,Y 569.847,Z 737.44,A -85,B 0,C 180,E1 2471.933,E2 2471.933} C_VEL
LIN {X 0,Y 569.932,Z 737.44,A -85,B 0,C 180,E1 2478.056,E2 2478.056} C_VEL
LIN {X 0,Y 569.95,Z 737.44,A -85,B 0,C 180,E1 2484.238,E2 2484.238} C_VEL
LIN {X 0,Y 569.975,Z 737.44,A -85,B 0,C 180,E1 2489.688,E2 2489.688} C_VEL
LIN {X 0,Y 570.117,Z 737.44,A -85,B 0,C 180,E1 2494.854,E2 2494.854} C_VEL
LIN {X 0,Y 570.175,Z 737.44,A -85,B 0,C 180,E1 2499.804,E2 2499.804} C_VEL
LIN {X 0,Y 570.03,Z 737.44,A -85,B 0,C 180,E1 2504.595,E2 2504.595} C_VEL
LIN {X 0,Y 570.146,Z 737.44,A -85,B 0,C 180,E1 2510.829,E2 2510.829} C_VEL
LIN {X 0,Y 570.232,Z 737.44,A -85,B 0,C 180,E1 2515.428,E2 2515.428} C_VEL
LIN {X 0,Y 570.26,Z 737.44,A -85,B 0,C 180,E1 2519.996,E2 2519.996} C_VEL
LIN {X 0,Y 570.307,Z 737.44,A -85,B 0,C 180,E1 2524.564,E2 2524.564} C_VEL
LIN {X 0,Y 570.288,Z 737.44,A -85,B 0,C 180,E1 2529.161,E2 2529.161} C_VEL
LIN {X 0,Y 570.228,Z 737.44,A -85,B 0,C 180,E1 2533.82,E2 2533.82} C_VEL
LIN {X 0,Y 570.192,Z 737.44,A -85,B 0,C 180,E1 2538.574,E2 2538.574} C_VEL
LIN {X 0,Y 570.128,Z 737.44,A -85,B 0,C 180,E1 2543.467,E2 2543.467} C_VEL
LIN {X 0,Y 569.963,Z 737.44,A -85,B 0,C 180,E1 2548.768,E2 2548.768} C_VEL
LIN {X 0,Y 569.945,Z 737.44,A -85,B 0,C 180,E1 2554.566,E2 2554.566} C_VEL
LIN {X 0,Y 569.889,Z 737.44,A -85,B 0,C 180,E1 2559.608,E2 2559.608} C_VEL
LIN {X 0,Y 569.937,Z 737.44,A -85,B 0,C 180,E1 2565.816,E2 2565.816} C_VEL
LIN {X 0,Y 569.954,Z 737.44,A -85,B 0,C 180,E1 2570.393,E2 2570.393} C_VEL
LIN {X 0,Y 569.877,Z 737.44,A -85,B 0,C 180,E1 2575.431,E2 2575.431} C_VEL
LIN {X 0,Y 569.947,Z 737.44,A -85,B 0,C 180,E1 2579.688,E2 2579.688} C_VEL
LIN {X 0,Y 570.024,Z 737.44,A -85,B 0,C 180,E1 2583.459,E2 2583.459} C_VEL
LIN {X 0,Y 574.596,Z 754.473,A -85,B 0,C 180,E1 2584.117,E2 2584.117} C_VEL
LIN {X 0,Y 574.018,Z 791.018,A -85,B 0,C 180,E1 2585.444,E2 2585.444} C_VEL
LIN {X 0,Y 573.161,Z 825.892,A -85,B 0,C 180,E1 2587.367,E2 2587.367} C_VEL
LIN {X 0,Y 572.271,Z 856.933,A -85,B 0,C 180,E1 2589.741,E2 2589.741} C_VEL
LIN {X 0,Y 571.547,Z 884.733,A -85,B 0,C 180,E1 2592.594,E2 2592.594} C_VEL
LIN {X 0,Y 571.059,Z 907.56,A -85,B 0,C 180,E1 2595.734,E2 2595.734} C_VEL
LIN {X 0,Y 570.763,Z 924.639,A -85,B 0,C 180,E1 2598.903,E2 2598.903} C_VEL
LIN {X 0,Y 570.569,Z 937.741,A -85,B 0,C 180,E1 2602.376,E2 2602.376} C_VEL
LIN {X 0,Y 570.53,Z 946.24,A -85,B 0,C 180,E1 2606.196,E2 2606.196} C_VEL
LIN {X 0,Y 570.504,Z 948.997,A -85,B 0,C 180,E1 2610,E2 2610} C_VEL
LIN {X 0,Y 570.532,Z 946.098,A -85,B 0,C 180,E1 2613.804,E2 2613.804} C_VEL
LIN {X 0,Y 570.605,Z 937.472,A -85,B 0,C 180,E1 2617.624,E2 2617.624} C_VEL
LIN {X 0,Y 570.808,Z 923.447,A -85,B 0,C 180,E1 2621.271,E2 2621.271} C_VEL
LIN {X 0,Y 571.176,Z 903.037,A -85,B 0,C 180,E1 2624.875,E2 2624.875} C_VEL
LIN {X 0,Y 571.732,Z 879.008,A -85,B 0,C 180,E1 2627.969,E2 2627.969} C_VEL
LIN {X 0,Y 572.511,Z 849.402,A -85,B 0,C 180,E1 2630.815,E2 2630.815} C_VEL
LIN {X 0,Y 573.385,Z 816.688,A -85,B 0,C 180,E1 2633.119,E2 2633.119} C_VEL
LIN {X 0,Y 574.186,Z 780.868,A -85,B 0,C 180,E1 2634.9,E2 2634.9} C_VEL
LIN {X 0,Y 573.892,Z 748.382,A -85,B 0,C 180,E1 2635.99,E2 2635.99} C_VEL
LIN {X 0,Y 570.317,Z 737.44,A -85,B 0,C 180,E1 2636.501,E2 2636.501} C_VEL
LIN {X 0,Y 570.029,Z 737.44,A -85,B 0,C 180,E1 2642.086,E2 2642.086} C_VEL
LIN {X 0,Y 569.876,Z 737.44,A -85,B 0,C 180,E1 2647.665,E2 2647.665} C_VEL
LIN {X 0,Y 569.865,Z 737.44,A -85,B 0,C 180,E1 2653.69,E2 2653.69} C_VEL
LIN {X 0,Y 569.953,Z 737.44,A -85,B 0,C 180,E1 2658.397,E2 2658.397} C_VEL
LIN {X 0,Y 569.932,Z 737.44,A -85,B 0,C 180,E1 2664.247,E2 2664.247} C_VEL
LIN {X 0,Y 569.969,Z 737.44,A -85,B 0,C 180,E1 2669.697,E2 2669.697} C_VEL
LIN {X 0,Y 570.107,Z 737.44,A -85,B 0,C 180,E1 2674.862,E2 2674.862} C_VEL
LIN {X 0,Y 570.224,Z 737.44,A -85,B 0,C 180,E1 2679.814,E2 2679.814} C_VEL
LIN {X 0,Y 570.384,Z 737.44,A -85,B 0,C 180,E1 2686.184,E2 2686.184} C_VEL
LIN {X 0,Y 570.322,Z 737.44,A -85,B 0,C 180,E1 2692.377,E2 2692.377} C_VEL
LIN {X 0,Y 570.376,Z 737.44,A -85,B 0,C 180,E1 2696.961,E2 2696.961} C_VEL
LIN {X 0,Y 570.484,Z 737.44,A -85,B 0,C 180,E1 2701.525,E2 2701.525} C_VEL
LIN {X 0,Y 570.445,Z 737.44,A -85,B 0,C 180,E1 2706.098,E2 2706.098} C_VEL
LIN {X 0,Y 570.222,Z 737.44,A -85,B 0,C 180,E1 2711.003,E2 2711.003} C_VEL
LIN {X 0,Y 566.159,Z 737.44,A -85,B 0,C 180,E1 2712.715,E2 2712.715} C_VEL
LIN {X 0,Y 562.171,Z 737.44,A -85,B 0,C 180,E1 2714.45,E2 2714.45} C_VEL
LIN {X 0,Y 562.21,Z 737.44,A -85,B 0,C 180,E1 2720.495,E2 2720.495} C_VEL
LIN {X 0,Y 562.22,Z 737.44,A -85,B 0,C 180,E1 2725.524,E2 2725.524} C_VEL
LIN {X 0,Y 562.02,Z 737.44,A -85,B 0,C 180,E1 2730.788,E2 2730.788} C_VEL
LIN {X 0,Y 562.048,Z 737.44,A -85,B 0,C 180,E1 2736.344,E2 2736.344} C_VEL
LIN {X 0,Y 562.004,Z 737.44,A -85,B 0,C 180,E1 2742.337,E2 2742.337} C_VEL
LIN {X 0,Y 561.924,Z 737.44,A -85,B 0,C 180,E1 2747.656,E2 2747.656} C_VEL
LIN {X 0,Y 562.117,Z 738.057,A -85,B 0,C 180,E1 2752.692,E2 2752.692} C_VEL
LIN {X 0,Y 571.507,Z 757.904,A -85,B 0,C 180,E1 2753.709,E2 2753.709} C_VEL
LIN {X 0,Y 571.223,Z 831.413,A -85,B 0,C 180,E1 2754.945,E2 2754.945} C_VEL
LIN {X 0,Y 570.305,Z 871.332,A -85,B 0,C 180,E1 2756.199,E2 2756.199} C_VEL
LIN {X 0,Y 569.01,Z 909.095,A -85,B 0,C 180,E1 2757.954,E2 2757.954} C_VEL
LIN {X 0,Y 567.392,Z 948.285,A -85,B 0,C 180,E1 2760.462,E2 2760.462} C_VEL
LIN {X 0,Y 565.777,Z 984.575,A -85,B 0,C 180,E1 2763.54,E2 2763.54} C_VEL
LIN {X 0,Y 564.551,Z 1015.361,A -85,B 0,C 180,E1 2766.908,E2 2766.908} C_VEL
LIN {X 0,Y 563.566,Z 1041.907,A -85,B 0,C 180,E1 2770.614,E2 2770.614} C_VEL
LIN {X 0,Y 563.009,Z 1064.306,A -85,B 0,C 180,E1 2774.713,E2 2774.713} C_VEL
LIN {X 0,Y 562.716,Z 1080.847,A -85,B 0,C 180,E1 2778.871,E2 2778.871} C_VEL
LIN {X 0,Y 562.654,Z 1090.332,A -85,B 0,C 180,E1 2782.268,E2 2782.268} C_VEL
LIN {X 0,Y 562.718,Z 1095.905,A -85,B 0,C 180,E1 2785.37,E2 2785.37} C_VEL
LIN {X 0,Y 562.684,Z 1098.657,A -85,B 0,C 180,E1 2788.458,E2 2788.458} C_VEL
LIN {X 0,Y 562.561,Z 1097.628,A -85,B 0,C 180,E1 2793.085,E2 2793.085} C_VEL
LIN {X 0,Y 562.728,Z 1091.918,A -85,B 0,C 180,E1 2796.954,E2 2796.954} C_VEL
LIN {X 0,Y 562.764,Z 1080.746,A -85,B 0,C 180,E1 2801.158,E2 2801.158} C_VEL
LIN {X 0,Y 563.085,Z 1064.24,A -85,B 0,C 180,E1 2805.298,E2 2805.298} C_VEL
LIN {X 0,Y 563.595,Z 1041.924,A -85,B 0,C 180,E1 2809.382,E2 2809.382} C_VEL
LIN {X 0,Y 564.61,Z 1013.693,A -85,B 0,C 180,E1 2813.298,E2 2813.298} C_VEL
LIN {X 0,Y 565.931,Z 981.4,A -85,B 0,C 180,E1 2816.763,E2 2816.763} C_VEL
LIN {X 0,Y 567.489,Z 946.278,A -85,B 0,C 180,E1 2819.687,E2 2819.687} C_VEL
LIN {X 0,Y 569.126,Z 906.295,A -85,B 0,C 180,E1 2822.199,E2 2822.199} C_VEL
LIN {X 0,Y 570.495,Z 865.942,A -85,B 0,C 180,E1 2824.009,E2 2824.009} C_VEL
LIN {X 0,Y 571.441,Z 826.259,A -85,B 0,C 180,E1 2825.162,E2 2825.162} C_VEL
LIN {X 0,Y 571.014,Z 756.184,A -85,B 0,C 180,E1 2826.353,E2 2826.353} C_VEL
LIN {X 0,Y 562.117,Z 738.056,A -85,B 0,C 180,E1 2827.308,E2 2827.308} C_VEL
LIN {X 0,Y 561.943,Z 737.44,A -85,B 0,C 180,E1 2833.327,E2 2833.327} C_VEL
LIN {X 0,Y 561.976,Z 737.44,A -85,B 0,C 180,E1 2838.967,E2 2838.967} C_VEL
LIN {X 0,Y 562.047,Z 737.44,A -85,B 0,C 180,E1 2843.912,E2 2843.912} C_VEL
LIN {X 0,Y 562.058,Z 737.44,A -85,B 0,C 180,E1 2849.538,E2 2849.538} C_VEL
LIN {X 0,Y 562.215,Z 737.44,A -85,B 0,C 180,E1 2854.475,E2 2854.475} C_VEL
LIN {X 0,Y 562.249,Z 737.44,A -85,B 0,C 180,E1 2860.468,E2 2860.468} C_VEL
LIN {X 0,Y 562.135,Z 737.44,A -85,B 0,C 180,E1 2864.373,E2 2864.373} C_VEL
LIN {X 0,Y 562.26,Z 737.44,A -85,B 0,C 180,E1 2870.699,E2 2870.699} C_VEL
LIN {X 0,Y 562.335,Z 737.44,A -85,B 0,C 180,E1 2875.364,E2 2875.364} C_VEL
LIN {X 0,Y 562.359,Z 737.44,A -85,B 0,C 180,E1 2879.996,E2 2879.996} C_VEL
LIN {X 0,Y 562.35,Z 737.44,A -85,B 0,C 180,E1 2885.041,E2 2885.041} C_VEL
LIN {X 0,Y 562.373,Z 737.44,A -85,B 0,C 180,E1 2889.291,E2 2889.291} C_VEL
LIN {X 0,Y 562.266,Z 737.44,A -85,B 0,C 180,E1 2894.221,E2 2894.221} C_VEL
LIN {X 0,Y 562.198,Z 737.44,A -85,B 0,C 180,E1 2899.517,E2 2899.517} C_VEL
LIN {X 0,Y 562.092,Z 737.44,A -85,B 0,C 180,E1 2905.522,E2 2905.522} C_VEL
LIN {X 0,Y 562.001,Z 737.44,A -85,B 0,C 180,E1 2910.779,E2 2910.779} C_VEL
LIN {X 0,Y 561.977,Z 737.44,A -85,B 0,C 180,E1 2916.34,E2 2916.34} C_VEL
LIN {X 0,Y 561.907,Z 737.44,A -85,B 0,C 180,E1 2922.335,E2 2922.335} C_VEL
LIN {X 0,Y 562.019,Z 737.44,A -85,B 0,C 180,E1 2927.666,E2 2927.666} C_VEL
LIN {X 0,Y 562.079,Z 737.44,A -85,B 0,C 180,E1 2933.894,E2 2933.894} C_VEL
LIN {X 0,Y 562.041,Z 737.44,A -85,B 0,C 180,E1 2939.526,E2 2939.526} C_VEL
LIN {X 0,Y 562.082,Z 737.798,A -85,B 0,C 180,E1 2943.08,E2 2943.08} C_VEL
LIN {X 0,Y 567.466,Z 755.694,A -85,B 0,C 180,E1 2943.801,E2 2943.801} C_VEL
LIN {X 0,Y 566.712,Z 793.086,A -85,B 0,C 180,E1 2945.209,E2 2945.209} C_VEL
LIN {X 0,Y 565.753,Z 825.878,A -85,B 0,C 180,E1 2947.054,E2 2947.054} C_VEL
LIN {X 0,Y 564.703,Z 857.406,A -85,B 0,C 180,E1 2949.5,E2 2949.5} C_VEL
LIN {X 0,Y 563.811,Z 886,A -85,B 0,C 180,E1 2952.507,E2 2952.507} C_VEL
LIN {X 0,Y 563.232,Z 908.37,A -85,B 0,C 180,E1 2955.665,E2 2955.665} C_VEL
LIN {X 0,Y 562.838,Z 926.425,A -85,B 0,C 180,E1 2959.147,E2 2959.147} C_VEL
LIN {X 0,Y 562.69,Z 938.886,A -85,B 0,C 180,E1 2962.657,E2 2962.657} C_VEL
LIN {X 0,Y 562.641,Z 946.239,A -85,B 0,C 180,E1 2966.143,E2 2966.143} C_VEL
LIN {X 0,Y 562.604,Z 948.997,A -85,B 0,C 180,E1 2970,E2 2970} C_VEL
LIN {X 0,Y 562.643,Z 946.1,A -85,B 0,C 180,E1 2973.857,E2 2973.857} C_VEL
LIN {X 0,Y 562.72,Z 938.62,A -85,B 0,C 180,E1 2977.342,E2 2977.342} C_VEL
LIN {X 0,Y 562.852,Z 926.027,A -85,B 0,C 180,E1 2980.853,E2 2980.853} C_VEL
LIN {X 0,Y 563.265,Z 907.781,A -85,B 0,C 180,E1 2984.341,E2 2984.341} C_VEL
LIN {X 0,Y 563.886,Z 883.903,A -85,B 0,C 180,E1 2987.663,E2 2987.663} C_VEL
LIN {X 0,Y 564.788,Z 855.255,A -85,B 0,C 180,E1 2990.6,E2 2990.6} C_VEL
LIN {X 0,Y 565.771,Z 824.466,A -85,B 0,C 180,E1 2992.951,E2 2992.951} C_VEL
LIN {X 0,Y 566.768,Z 788.693,A -85,B 0,C 180,E1 2994.907,E2 2994.907} C_VEL
LIN {X 0,Y 567.04,Z 751.707,A -85,B 0,C 180,E1 2996.238,E2 2996.238} C_VEL
LIN {X 0,Y 562.388,Z 737.44,A -85,B 0,C 180,E1 2996.896,E2 2996.896} C_VEL
LIN {X 0,Y 562.089,Z 737.44,A -85,B 0,C 180,E1 3003.4,E2 3003.4} C_VEL
LIN {X 0,Y 561.936,Z 737.44,A -85,B 0,C 180,E1 3008.63,E2 3008.63} C_VEL
LIN {X 0,Y 561.968,Z 737.44,A -85,B 0,C 180,E1 3014.464,E2 3014.464} C_VEL
LIN {X 0,Y 561.997,Z 737.44,A -85,B 0,C 180,E1 3019.727,E2 3019.727} C_VEL
LIN {X 0,Y 561.938,Z 737.44,A -85,B 0,C 180,E1 3025.551,E2 3025.551} C_VEL
LIN {X 0,Y 562.006,Z 737.44,A -85,B 0,C 180,E1 3031.001,E2 3031.001} C_VEL
LIN {X 0,Y 562.176,Z 737.44,A -85,B 0,C 180,E1 3036.299,E2 3036.299} C_VEL
LIN {X 0,Y 562.288,Z 737.44,A -85,B 0,C 180,E1 3041.155,E2 3041.155} C_VEL
LIN {X 0,Y 562.443,Z 737.44,A -85,B 0,C 180,E1 3045.985,E2 3045.985} C_VEL
LIN {X 0,Y 562.411,Z 737.44,A -85,B 0,C 180,E1 3052.269,E2 3052.269} C_VEL
LIN {X 0,Y 562.469,Z 737.44,A -85,B 0,C 180,E1 3056.918,E2 3056.918} C_VEL
LIN {X 0,Y 562.574,Z 737.44,A -85,B 0,C 180,E1 3061.546,E2 3061.546} C_VEL
LIN {X 0,Y 562.524,Z 737.44,A -85,B 0,C 180,E1 3066.184,E2 3066.184} C_VEL
LIN {X 0,Y 562.22,Z 737.44,A -85,B 0,C 180,E1 3072.444,E2 3072.444} C_VEL
LIN {X 0,Y 562.171,Z 737.44,A -85,B 0,C 180,E1 3074.45,E2 3074.45} C_VEL
LIN {X 0,Y 558.178,Z 737.44,A -85,B 0,C 180,E1 3076.192,E2 3076.192} C_VEL
LIN {X 0,Y 554.179,Z 737.44,A -85,B 0,C 180,E1 3077.959,E2 3077.959} C_VEL
LIN {X 0,Y 554.237,Z 737.44,A -85,B 0,C 180,E1 3082.487,E2 3082.487} C_VEL
LIN {X 0,Y 554.136,Z 737.44,A -85,B 0,C 180,E1 3087.678,E2 3087.678} C_VEL
LIN {X 0,Y 554.02,Z 737.44,A -85,B 0,C 180,E1 3093.132,E2 3093.132} C_VEL
LIN {X 0,Y 554.097,Z 737.44,A -85,B 0,C 180,E1 3098.937,E2 3098.937} C_VEL
LIN {X 0,Y 554.1,Z 737.44,A -85,B 0,C 180,E1 3104.732,E2 3104.732} C_VEL
LIN {X 0,Y 554.088,Z 737.44,A -85,B 0,C 180,E1 3111.064,E2 3111.064} C_VEL
LIN {X 0,Y 554.123,Z 737.538,A -85,B 0,C 180,E1 3112.051,E2 3112.051} C_VEL
LIN {X 0,Y 562.93,Z 755.806,A -85,B 0,C 180,E1 3113.033,E2 3113.033} C_VEL
LIN {X 0,Y 565.131,Z 760.08,A -85,B 0,C 180,E1 3113.267,E2 3113.267} C_VEL
LIN {X 0,Y 564.72,Z 832.523,A -85,B 0,C 180,E1 3114.507,E2 3114.507} C_VEL
LIN {X 0,Y 563.617,Z 872.818,A -85,B 0,C 180,E1 3115.805,E2 3115.805} C_VEL
LIN {X 0,Y 562.106,Z 909.835,A -85,B 0,C 180,E1 3117.558,E2 3117.558} C_VEL
LIN {X 0,Y 560.278,Z 948.199,A -85,B 0,C 180,E1 3120.042,E2 3120.042} C_VEL
LIN {X 0,Y 558.486,Z 984.168,A -85,B 0,C 180,E1 3123.126,E2 3123.126} C_VEL
LIN {X 0,Y 557.023,Z 1015.363,A -85,B 0,C 180,E1 3126.577,E2 3126.577} C_VEL
LIN {X 0,Y 555.871,Z 1042.31,A -85,B 0,C 180,E1 3130.402,E2 3130.402} C_VEL
LIN {X 0,Y 555.201,Z 1064.132,A -85,B 0,C 180,E1 3134.457,E2 3134.457} C_VEL
LIN {X 0,Y 554.851,Z 1080.439,A -85,B 0,C 180,E1 3138.59,E2 3138.59} C_VEL
LIN {X 0,Y 554.766,Z 1090.332,A -85,B 0,C 180,E1 3142.157,E2 3142.157} C_VEL
LIN {X 0,Y 554.82,Z 1095.905,A -85,B 0,C 180,E1 3145.304,E2 3145.304} C_VEL
LIN {X 0,Y 554.777,Z 1098.657,A -85,B 0,C 180,E1 3148.436,E2 3148.436} C_VEL
LIN {X 0,Y 554.672,Z 1097.628,A -85,B 0,C 180,E1 3153.129,E2 3153.129} C_VEL
LIN {X 0,Y 554.839,Z 1091.918,A -85,B 0,C 180,E1 3157.053,E2 3157.053} C_VEL
LIN {X 0,Y 554.895,Z 1081.778,A -85,B 0,C 180,E1 3161.01,E2 3161.01} C_VEL
LIN {X 0,Y 555.235,Z 1065.311,A -85,B 0,C 180,E1 3165.285,E2 3165.285} C_VEL
LIN {X 0,Y 555.869,Z 1042.345,A -85,B 0,C 180,E1 3169.592,E2 3169.592} C_VEL
LIN {X 0,Y 557.097,Z 1013.696,A -85,B 0,C 180,E1 3173.631,E2 3173.631} C_VEL
LIN {X 0,Y 558.623,Z 981.29,A -85,B 0,C 180,E1 3177.152,E2 3177.152} C_VEL
LIN {X 0,Y 560.442,Z 945.182,A -85,B 0,C 180,E1 3180.18,E2 3180.18} C_VEL
LIN {X 0,Y 562.309,Z 905.754,A -85,B 0,C 180,E1 3182.667,E2 3182.667} C_VEL
LIN {X 0,Y 563.909,Z 865.939,A -85,B 0,C 180,E1 3184.461,E2 3184.461} C_VEL
LIN {X 0,Y 564.953,Z 827.727,A -85,B 0,C 180,E1 3185.591,E2 3185.591} C_VEL
LIN {X 0,Y 564.685,Z 759.106,A -85,B 0,C 180,E1 3186.782,E2 3186.782} C_VEL
LIN {X 0,Y 554.24,Z 738.734,A -85,B 0,C 180,E1 3187.921,E2 3187.921} C_VEL
LIN {X 0,Y 554.131,Z 737.44,A -85,B 0,C 180,E1 3188.024,E2 3188.024} C_VEL
LIN {X 0,Y 554.044,Z 737.44,A -85,B 0,C 180,E1 3193.09,E2 3193.09} C_VEL
LIN {X 0,Y 554.077,Z 737.44,A -85,B 0,C 180,E1 3199.019,E2 3199.019} C_VEL
LIN {X 0,Y 554.06,Z 737.44,A -85,B 0,C 180,E1 3205.061,E2 3205.061} C_VEL
LIN {X 0,Y 554.141,Z 737.44,A -85,B 0,C 180,E1 3210.96,E2 3210.96} C_VEL
LIN {X 0,Y 554.239,Z 737.44,A -85,B 0,C 180,E1 3215.809,E2 3215.809} C_VEL
LIN {X 0,Y 554.357,Z 737.44,A -85,B 0,C 180,E1 3220.866,E2 3220.866} C_VEL
LIN {X 0,Y 554.077,Z 737.44,A -85,B 0,C 180,E1 3225.761,E2 3225.761} C_VEL
LIN {X 0,Y 554.349,Z 737.44,A -85,B 0,C 180,E1 3230.565,E2 3230.565} C_VEL
LIN {X 0,Y 554.46,Z 737.44,A -85,B 0,C 180,E1 3235.298,E2 3235.298} C_VEL
LIN {X 0,Y 554.459,Z 737.44,A -85,B 0,C 180,E1 3239.996,E2 3239.996} C_VEL
LIN {X 0,Y 554.501,Z 737.44,A -85,B 0,C 180,E1 3244.694,E2 3244.694} C_VEL
LIN {X 0,Y 554.346,Z 737.44,A -85,B 0,C 180,E1 3250.516,E2 3250.516} C_VEL
LIN {X 0,Y 554.233,Z 737.44,A -85,B 0,C 180,E1 3255.847,E2 3255.847} C_VEL
LIN {X 0,Y 554.258,Z 737.44,A -85,B 0,C 180,E1 3260.794,E2 3260.794} C_VEL
LIN {X 0,Y 554.147,Z 737.44,A -85,B 0,C 180,E1 3265.915,E2 3265.915} C_VEL
LIN {X 0,Y 554.063,Z 737.44,A -85,B 0,C 180,E1 3271.27,E2 3271.27} C_VEL
LIN {X 0,Y 553.989,Z 737.44,A -85,B 0,C 180,E1 3276.95,E2 3276.95} C_VEL
LIN {X 0,Y 554.029,Z 737.44,A -85,B 0,C 180,E1 3283.082,E2 3283.082} C_VEL
LIN {X 0,Y 554.096,Z 737.44,A -85,B 0,C 180,E1 3289.022,E2 3289.022} C_VEL
LIN {X 0,Y 554.079,Z 737.44,A -85,B 0,C 180,E1 3295.044,E2 3295.044} C_VEL
LIN {X 0,Y 554.071,Z 737.44,A -85,B 0,C 180,E1 3300.956,E2 3300.956} C_VEL
LIN {X 0,Y 554.1,Z 737.44,A -85,B 0,C 180,E1 3302.631,E2 3302.631} C_VEL
LIN {X 0,Y 560.356,Z 757.068,A -85,B 0,C 180,E1 3303.484,E2 3303.484} C_VEL
LIN {X 0,Y 559.469,Z 792.719,A -85,B 0,C 180,E1 3304.848,E2 3304.848} C_VEL
LIN {X 0,Y 558.356,Z 825.789,A -85,B 0,C 180,E1 3306.727,E2 3306.727} C_VEL
LIN {X 0,Y 557.167,Z 857.401,A -85,B 0,C 180,E1 3309.21,E2 3309.21} C_VEL
LIN {X 0,Y 556.171,Z 884.645,A -85,B 0,C 180,E1 3312.087,E2 3312.087} C_VEL
LIN {X 0,Y 555.437,Z 908.367,A -85,B 0,C 180,E1 3315.46,E2 3315.46} C_VEL
LIN {X 0,Y 554.972,Z 926.88,A -85,B 0,C 180,E1 3319.096,E2 3319.096} C_VEL
LIN {X 0,Y 554.793,Z 939.953,A -85,B 0,C 180,E1 3322.946,E2 3322.946} C_VEL
LIN {X 0,Y 554.704,Z 947.219,A -85,B 0,C 180,E1 3326.871,E2 3326.871} C_VEL
LIN {X 0,Y 554.734,Z 948.997,A -85,B 0,C 180,E1 3330,E2 3330} C_VEL
LIN {X 0,Y 554.771,Z 946.102,A -85,B 0,C 180,E1 3333.912,E2 3333.912} C_VEL
LIN {X 0,Y 554.855,Z 938.622,A -85,B 0,C 180,E1 3337.447,E2 3337.447} C_VEL
LIN {X 0,Y 554.999,Z 926.029,A -85,B 0,C 180,E1 3341.009,E2 3341.009} C_VEL
LIN {X 0,Y 555.471,Z 907.786,A -85,B 0,C 180,E1 3344.547,E2 3344.547} C_VEL
LIN {X 0,Y 556.203,Z 883.854,A -85,B 0,C 180,E1 3347.921,E2 3347.921} C_VEL
LIN {X 0,Y 557.267,Z 855.263,A -85,B 0,C 180,E1 3350.891,E2 3350.891} C_VEL
LIN {X 0,Y 558.447,Z 823.139,A -85,B 0,C 180,E1 3353.362,E2 3353.362} C_VEL
LIN {X 0,Y 559.515,Z 787.823,A -85,B 0,C 180,E1 3355.292,E2 3355.292} C_VEL
LIN {X 0,Y 559.965,Z 753.722,A -85,B 0,C 180,E1 3356.541,E2 3356.541} C_VEL
LIN {X 0,Y 554.414,Z 737.44,A -85,B 0,C 180,E1 3357.31,E2 3357.31} C_VEL
LIN {X 0,Y 554.175,Z 737.44,A -85,B 0,C 180,E1 3363.12,E2 3363.12} C_VEL
LIN {X 0,Y 554.013,Z 737.44,A -85,B 0,C 180,E1 3368.942,E2 3368.942} C_VEL
LIN {X 0,Y 554.111,Z 737.44,A -85,B 0,C 180,E1 3375.267,E2 3375.267} C_VEL
LIN {X 0,Y 554.081,Z 737.44,A -85,B 0,C 180,E1 3381.072,E2 3381.072} C_VEL
LIN {X 0,Y 554.007,Z 737.44,A -85,B 0,C 180,E1 3386.877,E2 3386.877} C_VEL
LIN {X 0,Y 554.14,Z 737.44,A -85,B 0,C 180,E1 3392.331,E2 3392.331} C_VEL
LIN {X 0,Y 554.255,Z 737.44,A -85,B 0,C 180,E1 3398.239,E2 3398.239} C_VEL
LIN {X 0,Y 554.403,Z 737.44,A -85,B 0,C 180,E1 3404.158,E2 3404.158} C_VEL
LIN {X 0,Y 554.383,Z 737.44,A -85,B 0,C 180,E1 3409.465,E2 3409.465} C_VEL
LIN {X 0,Y 554.51,Z 737.44,A -85,B 0,C 180,E1 3415.306,E2 3415.306} C_VEL
LIN {X 0,Y 554.664,Z 737.44,A -85,B 0,C 180,E1 3421.568,E2 3421.568} C_VEL
LIN {X 0,Y 554.595,Z 737.44,A -85,B 0,C 180,E1 3426.273,E2 3426.273} C_VEL
LIN {X 0,Y 554.297,Z 737.44,A -85,B 0,C 180,E1 3432.625,E2 3432.625} C_VEL
LIN {X 0,Y 554.179,Z 737.44,A -85,B 0,C 180,E1 3437.959,E2 3437.959} C_VEL
LIN {X 0,Y 550.276,Z 737.44,A -85,B 0,C 180,E1 3439.726,E2 3439.726} C_VEL
LIN {X 0,Y 546.308,Z 737.44,A -85,B 0,C 180,E1 3441.516,E2 3441.516} C_VEL
LIN {X 0,Y 546.291,Z 737.44,A -85,B 0,C 180,E1 3446.325,E2 3446.325} C_VEL
LIN {X 0,Y 546.116,Z 737.44,A -85,B 0,C 180,E1 3451.787,E2 3451.787} C_VEL
LIN {X 0,Y 546.169,Z 737.44,A -85,B 0,C 180,E1 3457.58,E2 3457.58} C_VEL
LIN {X 0,Y 546.166,Z 737.44,A -85,B 0,C 180,E1 3463.885,E2 3463.885} C_VEL
LIN {X 0,Y 546.156,Z 737.44,A -85,B 0,C 180,E1 3470.388,E2 3470.388} C_VEL
LIN {X 0,Y 546.209,Z 737.44,A -85,B 0,C 180,E1 3471.389,E2 3471.389} C_VEL
LIN {X 0,Y 551.103,Z 747.95,A -85,B 0,C 180,E1 3471.974,E2 3471.974} C_VEL
LIN {X 0,Y 558.779,Z 762.763,A -85,B 0,C 180,E1 3472.822,E2 3472.822} C_VEL
LIN {X 0,Y 558.254,Z 833.677,A -85,B 0,C 180,E1 3474.061,E2 3474.061} C_VEL
LIN {X 0,Y 556.936,Z 874.937,A -85,B 0,C 180,E1 3475.427,E2 3475.427} C_VEL
LIN {X 0,Y 555.179,Z 911.909,A -85,B 0,C 180,E1 3477.229,E2 3477.229} C_VEL
LIN {X 0,Y 553.116,Z 949.53,A -85,B 0,C 180,E1 3479.722,E2 3479.722} C_VEL
LIN {X 0,Y 551.094,Z 985.587,A -85,B 0,C 180,E1 3482.885,E2 3482.885} C_VEL
LIN {X 0,Y 549.397,Z 1016.976,A -85,B 0,C 180,E1 3486.448,E2 3486.448} C_VEL
LIN {X 0,Y 548.152,Z 1043.075,A -85,B 0,C 180,E1 3490.246,E2 3490.246} C_VEL
LIN {X 0,Y 547.387,Z 1064.724,A -85,B 0,C 180,E1 3494.356,E2 3494.356} C_VEL
LIN {X 0,Y 546.974,Z 1080.439,A -85,B 0,C 180,E1 3498.423,E2 3498.423} C_VEL
LIN {X 0,Y 546.897,Z 1090.332,A -85,B 0,C 180,E1 3502.044,E2 3502.044} C_VEL
LIN {X 0,Y 546.92,Z 1095.905,A -85,B 0,C 180,E1 3505.236,E2 3505.236} C_VEL
LIN {X 0,Y 546.872,Z 1098.657,A -85,B 0,C 180,E1 3508.413,E2 3508.413} C_VEL
LIN {X 0,Y 546.767,Z 1097.628,A -85,B 0,C 180,E1 3513.175,E2 3513.175} C_VEL
LIN {X 0,Y 546.943,Z 1091.918,A -85,B 0,C 180,E1 3517.155,E2 3517.155} C_VEL
LIN {X 0,Y 547.009,Z 1081.778,A -85,B 0,C 180,E1 3521.171,E2 3521.171} C_VEL
LIN {X 0,Y 547.406,Z 1064.724,A -85,B 0,C 180,E1 3525.644,E2 3525.644} C_VEL
LIN {X 0,Y 548.136,Z 1043.102,A -85,B 0,C 180,E1 3529.749,E2 3529.749} C_VEL
LIN {X 0,Y 549.504,Z 1015.366,A -85,B 0,C 180,E1 3533.762,E2 3533.762} C_VEL
LIN {X 0,Y 551.321,Z 982.076,A -85,B 0,C 180,E1 3537.466,E2 3537.466} C_VEL
LIN {X 0,Y 553.425,Z 945.185,A -85,B 0,C 180,E1 3540.603,E2 3540.603} C_VEL
LIN {X 0,Y 555.507,Z 905.757,A -85,B 0,C 180,E1 3543.118,E2 3543.118} C_VEL
LIN {X 0,Y 557.366,Z 864.612,A -85,B 0,C 180,E1 3544.98,E2 3544.98} C_VEL
LIN {X 0,Y 558.579,Z 826.087,A -85,B 0,C 180,E1 3546.101,E2 3546.101} C_VEL
LIN {X 0,Y 558.33,Z 761.841,A -85,B 0,C 180,E1 3547.228,E2 3547.228} C_VEL
LIN {X 0,Y 546.263,Z 738.347,A -85,B 0,C 180,E1 3548.582,E2 3548.582} C_VEL
LIN {X 0,Y 546.192,Z 737.44,A -85,B 0,C 180,E1 3548.736,E2 3548.736} C_VEL
LIN {X 0,Y 546.141,Z 737.44,A -85,B 0,C 180,E1 3553.882,E2 3553.882} C_VEL
LIN {X 0,Y 546.153,Z 737.44,A -85,B 0,C 180,E1 3558.457,E2 3558.457} C_VEL
LIN {X 0,Y 546.095,Z 737.44,A -85,B 0,C 180,E1 3564.393,E2 3564.393} C_VEL
LIN {X 0,Y 546.128,Z 737.44,A -85,B 0,C 180,E1 3570.064,E2 3570.064} C_VEL
LIN {X 0,Y 546.309,Z 737.44,A -85,B 0,C 180,E1 3576.139,E2 3576.139} C_VEL
LIN {X 0,Y 546.46,Z 737.44,A -85,B 0,C 180,E1 3582.253,E2 3582.253} C_VEL
LIN {X 0,Y 546.441,Z 737.44,A -85,B 0,C 180,E1 3588.814,E2 3588.814} C_VEL
LIN {X 0,Y 546.575,Z 737.44,A -85,B 0,C 180,E1 3595.23,E2 3595.23} C_VEL
LIN {X 0,Y 546.559,Z 737.44,A -85,B 0,C 180,E1 3599.996,E2 3599.996} C_VEL
LIN {X 0,Y 546.587,Z 737.44,A -85,B 0,C 180,E1 3604.762,E2 3604.762} C_VEL
LIN {X 0,Y 546.526,Z 737.44,A -85,B 0,C 180,E1 3609.563,E2 3609.563} C_VEL
LIN {X 0,Y 546.442,Z 737.44,A -85,B 0,C 180,E1 3614.434,E2 3614.434} C_VEL
LIN {X 0,Y 546.381,Z 737.44,A -85,B 0,C 180,E1 3619.59,E2 3619.59} C_VEL
LIN {X 0,Y 546.285,Z 737.44,A -85,B 0,C 180,E1 3624.558,E2 3624.558} C_VEL
LIN {X 0,Y 546.155,Z 737.44,A -85,B 0,C 180,E1 3629.925,E2 3629.925} C_VEL
LIN {X 0,Y 546.106,Z 737.44,A -85,B 0,C 180,E1 3635.596,E2 3635.596} C_VEL
LIN {X 0,Y 546.077,Z 737.44,A -85,B 0,C 180,E1 3641.703,E2 3641.703} C_VEL
LIN {X 0,Y 546.181,Z 737.44,A -85,B 0,C 180,E1 3646.133,E2 3646.133} C_VEL
LIN {X 0,Y 546.172,Z 737.44,A -85,B 0,C 180,E1 3652.422,E2 3652.422} C_VEL
LIN {X 0,Y 546.119,Z 737.44,A -85,B 0,C 180,E1 3658.215,E2 3658.215} C_VEL
LIN {X 0,Y 546.196,Z 737.44,A -85,B 0,C 180,E1 3662.218,E2 3662.218} C_VEL
LIN {X 0,Y 553.21,Z 759.707,A -85,B 0,C 180,E1 3663.203,E2 3663.203} C_VEL
LIN {X 0,Y 552.149,Z 795.614,A -85,B 0,C 180,E1 3664.639,E2 3664.639} C_VEL
LIN {X 0,Y 550.831,Z 829.967,A -85,B 0,C 180,E1 3666.684,E2 3666.684} C_VEL
LIN {X 0,Y 549.491,Z 860.529,A -85,B 0,C 180,E1 3669.205,E2 3669.205} C_VEL
LIN {X 0,Y 548.315,Z 888.48,A -85,B 0,C 180,E1 3672.318,E2 3672.318} C_VEL
LIN {X 0,Y 547.57,Z 911.586,A -85,B 0,C 180,E1 3675.795,E2 3675.795} C_VEL
LIN {X 0,Y 547.1,Z 928.893,A -85,B 0,C 180,E1 3679.44,E2 3679.44} C_VEL
LIN {X 0,Y 546.93,Z 939.952,A -85,B 0,C 180,E1 3682.844,E2 3682.844} C_VEL
LIN {X 0,Y 546.869,Z 946.238,A -85,B 0,C 180,E1 3686.031,E2 3686.031} C_VEL
LIN {X 0,Y 546.834,Z 948.997,A -85,B 0,C 180,E1 3690,E2 3690} C_VEL
LIN {X 0,Y 546.871,Z 946.103,A -85,B 0,C 180,E1 3693.969,E2 3693.969} C_VEL
LIN {X 0,Y 547.011,Z 937.478,A -85,B 0,C 180,E1 3697.955,E2 3697.955} C_VEL
LIN {X 0,Y 547.215,Z 924.289,A -85,B 0,C 180,E1 3701.571,E2 3701.571} C_VEL
LIN {X 0,Y 547.85,Z 904.643,A -85,B 0,C 180,E1 3705.277,E2 3705.277} C_VEL
LIN {X 0,Y 548.681,Z 881.127,A -85,B 0,C 180,E1 3708.501,E2 3708.501} C_VEL
LIN {X 0,Y 549.811,Z 852.969,A -85,B 0,C 180,E1 3711.399,E2 3711.399} C_VEL
LIN {X 0,Y 551.221,Z 820.673,A -85,B 0,C 180,E1 3713.854,E2 3713.854} C_VEL
LIN {X 0,Y 552.427,Z 785.509,A -85,B 0,C 180,E1 3715.745,E2 3715.745} C_VEL
LIN {X 0,Y 552.581,Z 754.995,A -85,B 0,C 180,E1 3716.889,E2 3716.889} C_VEL
LIN {X 0,Y 546.452,Z 737.44,A -85,B 0,C 180,E1 3717.73,E2 3717.73} C_VEL
LIN {X 0,Y 546.199,Z 737.44,A -85,B 0,C 180,E1 3723.755,E2 3723.755} C_VEL
LIN {X 0,Y 546.093,Z 737.44,A -85,B 0,C 180,E1 3729.617,E2 3729.617} C_VEL
LIN {X 0,Y 546.161,Z 737.44,A -85,B 0,C 180,E1 3736.141,E2 3736.141} C_VEL
LIN {X 0,Y 546.152,Z 737.44,A -85,B 0,C 180,E1 3742.429,E2 3742.429} C_VEL
LIN {X 0,Y 546.108,Z 737.44,A -85,B 0,C 180,E1 3748.222,E2 3748.222} C_VEL
LIN {X 0,Y 546.285,Z 737.44,A -85,B 0,C 180,E1 3753.684,E2 3753.684} C_VEL
LIN {X 0,Y 546.412,Z 737.44,A -85,B 0,C 180,E1 3758.894,E2 3758.894} C_VEL
LIN {X 0,Y 546.501,Z 737.44,A -85,B 0,C 180,E1 3763.922,E2 3763.922} C_VEL
LIN {X 0,Y 546.489,Z 737.44,A -85,B 0,C 180,E1 3768.823,E2 3768.823} C_VEL
LIN {X 0,Y 546.489,Z 737.44,A -85,B 0,C 180,E1 3773.642,E2 3773.642} C_VEL
LIN {X 0,Y 546.49,Z 737.44,A -85,B 0,C 180,E1 3778.417,E2 3778.417} C_VEL
LIN {X 0,Y 546.498,Z 737.44,A -85,B 0,C 180,E1 3783.18,E2 3783.18} C_VEL
LIN {X 0,Y 546.426,Z 737.44,A -85,B 0,C 180,E1 3787.967,E2 3787.967} C_VEL
LIN {X 0,Y 546.376,Z 737.44,A -85,B 0,C 180,E1 3792.811,E2 3792.811} C_VEL
LIN {X 0,Y 546.272,Z 737.44,A -85,B 0,C 180,E1 3797.95,E2 3797.95} C_VEL
LIN {X 0,Y 546.308,Z 737.44,A -85,B 0,C 180,E1 3801.516,E2 3801.516} C_VEL
LIN {X 0,Y 542.325,Z 737.44,A -85,B 0,C 180,E1 3803.306,E2 3803.306} C_VEL
LIN {X 0,Y 538.371,Z 737.44,A -85,B 0,C 180,E1 3805.121,E2 3805.121} C_VEL
LIN {X 0,Y 538.215,Z 737.44,A -85,B 0,C 180,E1 3810.422,E2 3810.422} C_VEL
LIN {X 0,Y 538.195,Z 737.44,A -85,B 0,C 180,E1 3816.212,E2 3816.212} C_VEL
LIN {X 0,Y 538.174,Z 737.44,A -85,B 0,C 180,E1 3822.469,E2 3822.469} C_VEL
LIN {X 0,Y 538.126,Z 737.44,A -85,B 0,C 180,E1 3827.528,E2 3827.528} C_VEL
LIN {X 0,Y 538.293,Z 737.678,A -85,B 0,C 180,E1 3830.727,E2 3830.727} C_VEL
LIN {X 0,Y 544.909,Z 751.399,A -85,B 0,C 180,E1 3831.52,E2 3831.52} C_VEL
LIN {X 0,Y 552.523,Z 767.205,A -85,B 0,C 180,E1 3832.4,E2 3832.4} C_VEL
LIN {X 0,Y 551.836,Z 834.409,A -85,B 0,C 180,E1 3833.594,E2 3833.594} C_VEL
LIN {X 0,Y 550.321,Z 875.488,A -85,B 0,C 180,E1 3834.974,E2 3834.974} C_VEL
LIN {X 0,Y 548.342,Z 912.673,A -85,B 0,C 180,E1 3836.816,E2 3836.816} C_VEL
LIN {X 0,Y 546.059,Z 949.763,A -85,B 0,C 180,E1 3839.309,E2 3839.309} C_VEL
LIN {X 0,Y 543.912,Z 984.02,A -85,B 0,C 180,E1 3842.329,E2 3842.329} C_VEL
LIN {X 0,Y 541.96,Z 1015.365,A -85,B 0,C 180,E1 3845.886,E2 3845.886} C_VEL
LIN {X 0,Y 540.483,Z 1043.077,A -85,B 0,C 180,E1 3849.954,E2 3849.954} C_VEL
LIN {X 0,Y 539.605,Z 1064.722,A -85,B 0,C 180,E1 3854.124,E2 3854.124} C_VEL
LIN {X 0,Y 539.1,Z 1081.776,A -85,B 0,C 180,E1 3858.663,E2 3858.663} C_VEL
LIN {X 0,Y 538.943,Z 1091.918,A -85,B 0,C 180,E1 3862.738,E2 3862.738} C_VEL
LIN {X 0,Y 538.871,Z 1097.627,A -85,B 0,C 180,E1 3866.779,E2 3866.779} C_VEL
LIN {X 0,Y 538.853,Z 1099,A -85,B 0,C 180,E1 3870,E2 3870} C_VEL
LIN {X 0,Y 538.881,Z 1097.628,A -85,B 0,C 180,E1 3873.221,E2 3873.221} C_VEL
LIN {X 0,Y 539.042,Z 1091.918,A -85,B 0,C 180,E1 3877.261,E2 3877.261} C_VEL
LIN {X 0,Y 539.132,Z 1081.777,A -85,B 0,C 180,E1 3881.337,E2 3881.337} C_VEL
LIN {X 0,Y 539.58,Z 1064.721,A -85,B 0,C 180,E1 3885.877,E2 3885.877} C_VEL
LIN {X 0,Y 540.549,Z 1041.953,A -85,B 0,C 180,E1 3890.238,E2 3890.238} C_VEL
LIN {X 0,Y 542.041,Z 1013.689,A -85,B 0,C 180,E1 3894.33,E2 3894.33} C_VEL
LIN {X 0,Y 544.071,Z 982.194,A -85,B 0,C 180,E1 3897.852,E2 3897.852} C_VEL
LIN {X 0,Y 546.454,Z 945.171,A -85,B 0,C 180,E1 3901.038,E2 3901.038} C_VEL
LIN {X 0,Y 548.745,Z 906.251,A -85,B 0,C 180,E1 3903.552,E2 3903.552} C_VEL
LIN {X 0,Y 550.765,Z 865.796,A -85,B 0,C 180,E1 3905.411,E2 3905.411} C_VEL
LIN {X 0,Y 552.093,Z 828.004,A -85,B 0,C 180,E1 3906.545,E2 3906.545} C_VEL
LIN {X 0,Y 552.017,Z 764.952,A -85,B 0,C 180,E1 3907.677,E2 3907.677} C_VEL
LIN {X 0,Y 538.444,Z 739.09,A -85,B 0,C 180,E1 3909.236,E2 3909.236} C_VEL
LIN {X 0,Y 538.287,Z 737.44,A -85,B 0,C 180,E1 3909.349,E2 3909.349} C_VEL
LIN {X 0,Y 538.188,Z 737.44,A -85,B 0,C 180,E1 3915.308,E2 3915.308} C_VEL
LIN {X 0,Y 538.226,Z 737.44,A -85,B 0,C 180,E1 3921.767,E2 3921.767} C_VEL
LIN {X 0,Y 538.15,Z 737.44,A -85,B 0,C 180,E1 3927.686,E2 3927.686} C_VEL
LIN {X 0,Y 538.357,Z 737.44,A -85,B 0,C 180,E1 3933.257,E2 3933.257} C_VEL
LIN {X 0,Y 538.434,Z 737.44,A -85,B 0,C 180,E1 3938.557,E2 3938.557} C_VEL
LIN {X 0,Y 538.466,Z 737.44,A -85,B 0,C 180,E1 3943.667,E2 3943.667} C_VEL
LIN {X 0,Y 538.531,Z 737.44,A -85,B 0,C 180,E1 3950.285,E2 3950.285} C_VEL
LIN {X 0,Y 538.672,Z 737.44,A -85,B 0,C 180,E1 3955.159,E2 3955.159} C_VEL
LIN {X 0,Y 538.677,Z 737.44,A -85,B 0,C 180,E1 3959.996,E2 3959.996} C_VEL
LIN {X 0,Y 538.674,Z 737.44,A -85,B 0,C 180,E1 3964.832,E2 3964.832} C_VEL
LIN {X 0,Y 538.537,Z 737.44,A -85,B 0,C 180,E1 3970.278,E2 3970.278} C_VEL
LIN {X 0,Y 538.439,Z 737.44,A -85,B 0,C 180,E1 3976.325,E2 3976.325} C_VEL
LIN {X 0,Y 538.382,Z 737.44,A -85,B 0,C 180,E1 3981.876,E2 3981.876} C_VEL
LIN {X 0,Y 538.303,Z 737.44,A -85,B 0,C 180,E1 3986.737,E2 3986.737} C_VEL
LIN {X 0,Y 538.23,Z 737.44,A -85,B 0,C 180,E1 3992.449,E2 3992.449} C_VEL
LIN {X 0,Y 538.161,Z 737.44,A -85,B 0,C 180,E1 3998.228,E2 3998.228} C_VEL
LIN {X 0,Y 538.185,Z 737.44,A -85,B 0,C 180,E1 4004.681,E2 4004.681} C_VEL
LIN {X 0,Y 538.193,Z 737.44,A -85,B 0,C 180,E1 4009.683,E2 4009.683} C_VEL
LIN {X 0,Y 538.154,Z 737.44,A -85,B 0,C 180,E1 4015.76,E2 4015.76} C_VEL
LIN {X 0,Y 538.254,Z 737.494,A -85,B 0,C 180,E1 4021.78,E2 4021.78} C_VEL
LIN {X 0,Y 546.095,Z 761.569,A -85,B 0,C 180,E1 4022.889,E2 4022.889} C_VEL
LIN {X 0,Y 544.902,Z 797.033,A -85,B 0,C 180,E1 4024.351,E2 4024.351} C_VEL
LIN {X 0,Y 543.381,Z 831.725,A -85,B 0,C 180,E1 4026.474,E2 4026.474} C_VEL
LIN {X 0,Y 541.877,Z 862.101,A -85,B 0,C 180,E1 4029.06,E2 4029.06} C_VEL
LIN {X 0,Y 540.592,Z 889.456,A -85,B 0,C 180,E1 4032.186,E2 4032.186} C_VEL
LIN {X 0,Y 539.743,Z 912.683,A -85,B 0,C 180,E1 4035.792,E2 4035.792} C_VEL
LIN {X 0,Y 539.248,Z 928.823,A -85,B 0,C 180,E1 4039.267,E2 4039.267} C_VEL
LIN {X 0,Y 539.039,Z 939.95,A -85,B 0,C 180,E1 4042.739,E2 4042.739} C_VEL
LIN {X 0,Y 538.957,Z 946.462,A -85,B 0,C 180,E1 4046.125,E2 4046.125} C_VEL
LIN {X 0,Y 538.939,Z 948.997,A -85,B 0,C 180,E1 4050,E2 4050} C_VEL
LIN {X 0,Y 538.96,Z 946.326,A -85,B 0,C 180,E1 4053.878,E2 4053.878} C_VEL
LIN {X 0,Y 539.1,Z 938.626,A -85,B 0,C 180,E1 4057.666,E2 4057.666} C_VEL
LIN {X 0,Y 539.306,Z 926.034,A -85,B 0,C 180,E1 4061.333,E2 4061.333} C_VEL
LIN {X 0,Y 539.903,Z 908.303,A -85,B 0,C 180,E1 4064.888,E2 4064.888} C_VEL
LIN {X 0,Y 540.858,Z 884.583,A -85,B 0,C 180,E1 4068.356,E2 4068.356} C_VEL
LIN {X 0,Y 542.191,Z 856.425,A -85,B 0,C 180,E1 4071.392,E2 4071.392} C_VEL
LIN {X 0,Y 543.676,Z 824.733,A -85,B 0,C 180,E1 4073.923,E2 4073.923} C_VEL
LIN {X 0,Y 545.128,Z 788.763,A -85,B 0,C 180,E1 4075.968,E2 4075.968} C_VEL
LIN {X 0,Y 545.574,Z 757.432,A -85,B 0,C 180,E1 4077.19,E2 4077.19} C_VEL
LIN {X 0,Y 538.474,Z 737.44,A -85,B 0,C 180,E1 4078.161,E2 4078.161} C_VEL
LIN {X 0,Y 538.241,Z 737.44,A -85,B 0,C 180,E1 4084.234,E2 4084.234} C_VEL
LIN {X 0,Y 538.108,Z 737.44,A -85,B 0,C 180,E1 4090.578,E2 4090.578} C_VEL
LIN {X 0,Y 538.199,Z 737.44,A -85,B 0,C 180,E1 4097.004,E2 4097.004} C_VEL
LIN {X 0,Y 538.219,Z 737.44,A -85,B 0,C 180,E1 4101.965,E2 4101.965} C_VEL
LIN {X 0,Y 538.138,Z 737.44,A -85,B 0,C 180,E1 4107.695,E2 4107.695} C_VEL
LIN {X 0,Y 538.353,Z 737.44,A -85,B 0,C 180,E1 4113.266,E2 4113.266} C_VEL
LIN {X 0,Y 538.452,Z 737.44,A -85,B 0,C 180,E1 4118.566,E2 4118.566} C_VEL
LIN {X 0,Y 538.563,Z 737.44,A -85,B 0,C 180,E1 4123.679,E2 4123.679} C_VEL
LIN {X 0,Y 538.606,Z 737.44,A -85,B 0,C 180,E1 4129.683,E2 4129.683} C_VEL
LIN {X 0,Y 538.68,Z 737.44,A -85,B 0,C 180,E1 4135.168,E2 4135.168} C_VEL
LIN {X 0,Y 538.864,Z 737.44,A -85,B 0,C 180,E1 4141.614,E2 4141.614} C_VEL
LIN {X 0,Y 538.757,Z 737.44,A -85,B 0,C 180,E1 4146.458,E2 4146.458} C_VEL
LIN {X 0,Y 538.585,Z 737.44,A -85,B 0,C 180,E1 4151.352,E2 4151.352} C_VEL
LIN {X 0,Y 538.375,Z 737.44,A -85,B 0,C 180,E1 4157.034,E2 4157.034} C_VEL
LIN {X 0,Y 538.383,Z 737.44,A -85,B 0,C 180,E1 4161.875,E2 4161.875} C_VEL
LIN {X 0,Y 538.371,Z 737.44,A -85,B 0,C 180,E1 4165.121,E2 4165.121} C_VEL
LIN {X 0,Y 537.052,Z 737.44,A -85,B 0,C 180,E1 4166.043,E2 4166.043} C_VEL
LIN {X 0,Y 530.379,Z 737.44,A -85,B 0,C 180,E1 4168.553,E2 4168.553} C_VEL
LIN {X 0,Y 530.298,Z 737.44,A -85,B 0,C 180,E1 4168.791,E2 4168.791} C_VEL
LIN {X 0,Y 530.255,Z 737.44,A -85,B 0,C 180,E1 4174.825,E2 4174.825} C_VEL
LIN {X 0,Y 530.263,Z 737.44,A -85,B 0,C 180,E1 4181.049,E2 4181.049} C_VEL
LIN {X 0,Y 530.253,Z 737.44,A -85,B 0,C 180,E1 4186.744,E2 4186.744} C_VEL
LIN {X 0,Y 530.352,Z 738.174,A -85,B 0,C 180,E1 4190.031,E2 4190.031} C_VEL
LIN {X 0,Y 546.268,Z 769.264,A -85,B 0,C 180,E1 4191.926,E2 4191.926} C_VEL
LIN {X 0,Y 545.44,Z 834.617,A -85,B 0,C 180,E1 4193.103,E2 4193.103} C_VEL
LIN {X 0,Y 543.766,Z 875.92,A -85,B 0,C 180,E1 4194.508,E2 4194.508} C_VEL
LIN {X 0,Y 541.49,Z 914.388,A -85,B 0,C 180,E1 4196.449,E2 4196.449} C_VEL
LIN {X 0,Y 538.92,Z 951.635,A -85,B 0,C 180,E1 4199.015,E2 4199.015} C_VEL
LIN {X 0,Y 536.457,Z 986.509,A -85,B 0,C 180,E1 4202.182,E2 4202.182} C_VEL
LIN {X 0,Y 534.347,Z 1017.236,A -85,B 0,C 180,E1 4205.778,E2 4205.778} C_VEL
LIN {X 0,Y 532.758,Z 1043.957,A -85,B 0,C 180,E1 4209.807,E2 4209.807} C_VEL
LIN {X 0,Y 531.839,Z 1064.721,A -85,B 0,C 180,E1 4213.886,E2 4213.886} C_VEL
LIN {X 0,Y 531.226,Z 1081.775,A -85,B 0,C 180,E1 4218.492,E2 4218.492} C_VEL
LIN {X 0,Y 531.06,Z 1091.918,A -85,B 0,C 180,E1 4222.629,E2 4222.629} C_VEL
LIN {X 0,Y 530.984,Z 1097.627,A -85,B 0,C 180,E1 4226.731,E2 4226.731} C_VEL
LIN {X 0,Y 530.953,Z 1099,A -85,B 0,C 180,E1 4230,E2 4230} C_VEL
LIN {X 0,Y 530.962,Z 1097.248,A -85,B 0,C 180,E1 4233.637,E2 4233.637} C_VEL
LIN {X 0,Y 531.103,Z 1090.332,A -85,B 0,C 180,E1 4238.194,E2 4238.194} C_VEL
LIN {X 0,Y 531.271,Z 1079.094,A -85,B 0,C 180,E1 4242.341,E2 4242.341} C_VEL
LIN {X 0,Y 531.846,Z 1062.773,A -85,B 0,C 180,E1 4246.539,E2 4246.539} C_VEL
LIN {X 0,Y 532.953,Z 1040.859,A -85,B 0,C 180,E1 4250.719,E2 4250.719} C_VEL
LIN {X 0,Y 534.599,Z 1013.152,A -85,B 0,C 180,E1 4254.759,E2 4254.759} C_VEL
LIN {X 0,Y 536.824,Z 981.737,A -85,B 0,C 180,E1 4258.307,E2 4258.307} C_VEL
LIN {X 0,Y 539.44,Z 945.734,A -85,B 0,C 180,E1 4261.443,E2 4261.443} C_VEL
LIN {X 0,Y 542.05,Z 906.254,A -85,B 0,C 180,E1 4264.023,E2 4264.023} C_VEL
LIN {X 0,Y 544.364,Z 865.078,A -85,B 0,C 180,E1 4265.923,E2 4265.923} C_VEL
LIN {X 0,Y 545.806,Z 827.08,A -85,B 0,C 180,E1 4267.06,E2 4267.06} C_VEL
LIN {X 0,Y 545.868,Z 768.048,A -85,B 0,C 180,E1 4268.126,E2 4268.126} C_VEL
LIN {X 0,Y 530.347,Z 738.247,A -85,B 0,C 180,E1 4269.969,E2 4269.969} C_VEL
LIN {X 0,Y 530.259,Z 737.44,A -85,B 0,C 180,E1 4274.454,E2 4274.454} C_VEL
LIN {X 0,Y 530.226,Z 737.44,A -85,B 0,C 180,E1 4280.439,E2 4280.439} C_VEL
LIN {X 0,Y 530.248,Z 737.44,A -85,B 0,C 180,E1 4285.896,E2 4285.896} C_VEL
LIN {X 0,Y 530.331,Z 737.44,A -85,B 0,C 180,E1 4292.25,E2 4292.25} C_VEL
LIN {X 0,Y 530.523,Z 737.44,A -85,B 0,C 180,E1 4298.221,E2 4298.221} C_VEL
LIN {X 0,Y 530.568,Z 737.44,A -85,B 0,C 180,E1 4303.417,E2 4303.417} C_VEL
LIN {X 0,Y 530.636,Z 737.44,A -85,B 0,C 180,E1 4310.139,E2 4310.139} C_VEL
LIN {X 0,Y 530.768,Z 737.44,A -85,B 0,C 180,E1 4315.087,E2 4315.087} C_VEL
LIN {X 0,Y 530.777,Z 737.44,A -85,B 0,C 180,E1 4319.996,E2 4319.996} C_VEL
LIN {X 0,Y 530.761,Z 737.44,A -85,B 0,C 180,E1 4324.904,E2 4324.904} C_VEL
LIN {X 0,Y 530.694,Z 737.44,A -85,B 0,C 180,E1 4329.851,E2 4329.851} C_VEL
LIN {X 0,Y 530.586,Z 737.44,A -85,B 0,C 180,E1 4334.875,E2 4334.875} C_VEL
LIN {X 0,Y 530.53,Z 737.44,A -85,B 0,C 180,E1 4340.02,E2 4340.02} C_VEL
LIN {X 0,Y 530.415,Z 737.44,A -85,B 0,C 180,E1 4345.343,E2 4345.343} C_VEL
LIN {X 0,Y 530.273,Z 737.44,A -85,B 0,C 180,E1 4351.071,E2 4351.071} C_VEL
LIN {X 0,Y 530.204,Z 737.44,A -85,B 0,C 180,E1 4356.914,E2 4356.914} C_VEL
LIN {X 0,Y 530.252,Z 737.44,A -85,B 0,C 180,E1 4363.245,E2 4363.245} C_VEL
LIN {X 0,Y 530.263,Z 737.44,A -85,B 0,C 180,E1 4368.952,E2 4368.952} C_VEL
LIN {X 0,Y 530.257,Z 737.44,A -85,B 0,C 180,E1 4375.177,E2 4375.177} C_VEL
LIN {X 0,Y 530.275,Z 737.454,A -85,B 0,C 180,E1 4381.251,E2 4381.251} C_VEL
LIN {X 0,Y 538.947,Z 764.243,A -85,B 0,C 180,E1 4382.593,E2 4382.593} C_VEL
LIN {X 0,Y 537.605,Z 799.919,A -85,B 0,C 180,E1 4384.13,E2 4384.13} C_VEL
LIN {X 0,Y 535.932,Z 833.412,A -85,B 0,C 180,E1 4386.262,E2 4386.262} C_VEL
LIN {X 0,Y 534.2,Z 864.34,A -85,B 0,C 180,E1 4388.977,E2 4388.977} C_VEL
LIN {X 0,Y 532.825,Z 891.937,A -85,B 0,C 180,E1 4392.256,E2 4392.256} C_VEL
LIN {X 0,Y 531.907,Z 913.402,A -85,B 0,C 180,E1 4395.717,E2 4395.717} C_VEL
LIN {X 0,Y 531.371,Z 928.821,A -85,B 0,C 180,E1 4399.106,E2 4399.106} C_VEL
LIN {X 0,Y 531.165,Z 939.948,A -85,B 0,C 180,E1 4402.631,E2 4402.631} C_VEL
LIN {X 0,Y 531.058,Z 946.476,A -85,B 0,C 180,E1 4406.076,E2 4406.076} C_VEL
LIN {X 0,Y 531.039,Z 948.997,A -85,B 0,C 180,E1 4410,E2 4410} C_VEL
LIN {X 0,Y 531.064,Z 946.331,A -85,B 0,C 180,E1 4413.933,E2 4413.933} C_VEL
LIN {X 0,Y 531.24,Z 938.628,A -85,B 0,C 180,E1 4417.78,E2 4417.78} C_VEL
LIN {X 0,Y 531.458,Z 926.036,A -85,B 0,C 180,E1 4421.503,E2 4421.503} C_VEL
LIN {X 0,Y 532.194,Z 907.463,A -85,B 0,C 180,E1 4425.257,E2 4425.257} C_VEL
LIN {X 0,Y 533.31,Z 882.887,A -85,B 0,C 180,E1 4428.84,E2 4428.84} C_VEL
LIN {X 0,Y 534.722,Z 855.338,A -85,B 0,C 180,E1 4431.81,E2 4431.81} C_VEL
LIN {X 0,Y 536.35,Z 824.73,A -85,B 0,C 180,E1 4434.272,E2 4434.272} C_VEL
LIN {X 0,Y 537.995,Z 788.698,A -85,B 0,C 180,E1 4436.342,E2 4436.342} C_VEL
LIN {X 0,Y 538.542,Z 759.909,A -85,B 0,C 180,E1 4437.489,E2 4437.489} C_VEL
LIN {X 0,Y 530.48,Z 737.44,A -85,B 0,C 180,E1 4438.714,E2 4438.714} C_VEL
LIN {X 0,Y 530.306,Z 737.44,A -85,B 0,C 180,E1 4444.819,E2 4444.819} C_VEL
LIN {X 0,Y 530.158,Z 737.44,A -85,B 0,C 180,E1 4451.058,E2 4451.058} C_VEL
LIN {X 0,Y 530.293,Z 737.44,A -85,B 0,C 180,E1 4456.759,E2 4456.759} C_VEL
LIN {X 0,Y 530.227,Z 737.44,A -85,B 0,C 180,E1 4463.083,E2 4463.083} C_VEL
LIN {X 0,Y 530.239,Z 737.44,A -85,B 0,C 180,E1 4469.08,E2 4469.08} C_VEL
LIN {X 0,Y 530.48,Z 737.44,A -85,B 0,C 180,E1 4474.66,E2 4474.66} C_VEL
LIN {X 0,Y 530.646,Z 737.44,A -85,B 0,C 180,E1 4480.31,E2 4480.31} C_VEL
LIN {X 0,Y 530.711,Z 737.44,A -85,B 0,C 180,E1 4485.916,E2 4485.916} C_VEL
LIN {X 0,Y 530.767,Z 737.44,A -85,B 0,C 180,E1 4491.805,E2 4491.805} C_VEL
LIN {X 0,Y 530.86,Z 737.44,A -85,B 0,C 180,E1 4496.735,E2 4496.735} C_VEL
LIN {X 0,Y 530.954,Z 737.44,A -85,B 0,C 180,E1 4501.638,E2 4501.638} C_VEL
LIN {X 0,Y 530.844,Z 737.44,A -85,B 0,C 180,E1 4506.554,E2 4506.554} C_VEL
LIN {X 0,Y 530.653,Z 737.44,A -85,B 0,C 180,E1 4511.524,E2 4511.524} C_VEL
LIN {X 0,Y 530.511,Z 737.44,A -85,B 0,C 180,E1 4516.585,E2 4516.585} C_VEL
LIN {X 0,Y 530.512,Z 737.44,A -85,B 0,C 180,E1 4521.78,E2 4521.78} C_VEL
LIN {X 0,Y 530.331,Z 737.44,A -85,B 0,C 180,E1 4527.75,E2 4527.75} C_VEL
LIN {X 0,Y 530.298,Z 737.44,A -85,B 0,C 180,E1 4528.791,E2 4528.791} C_VEL
LIN {X 0,Y 527.759,Z 737.44,A -85,B 0,C 180,E1 4530.179,E2 4530.179} C_VEL
LIN {X 0,Y 522.376,Z 737.44,A -85,B 0,C 180,E1 4532.259,E2 4532.259} C_VEL
LIN {X 0,Y 522.3,Z 737.44,A -85,B 0,C 180,E1 4532.5,E2 4532.5} C_VEL
LIN {X 0,Y 522.299,Z 737.44,A -85,B 0,C 180,E1 4538.496,E2 4538.496} C_VEL
LIN {X 0,Y 522.347,Z 737.44,A -85,B 0,C 180,E1 4544.079,E2 4544.079} C_VEL
LIN {X 0,Y 522.335,Z 737.44,A -85,B 0,C 180,E1 4549.294,E2 4549.294} C_VEL
LIN {X 0,Y 526.395,Z 746.493,A -85,B 0,C 180,E1 4549.814,E2 4549.814} C_VEL
LIN {X 0,Y 540.032,Z 771.538,A -85,B 0,C 180,E1 4551.444,E2 4551.444} C_VEL
LIN {X 0,Y 539.082,Z 835.176,A -85,B 0,C 180,E1 4552.61,E2 4552.61} C_VEL
LIN {X 0,Y 537.221,Z 876.514,A -85,B 0,C 180,E1 4554.035,E2 4554.035} C_VEL
LIN {X 0,Y 534.696,Z 915.478,A -85,B 0,C 180,E1 4556.035,E2 4556.035} C_VEL
LIN {X 0,Y 531.865,Z 952.666,A -85,B 0,C 180,E1 4558.647,E2 4558.647} C_VEL
LIN {X 0,Y 529.171,Z 987.11,A -85,B 0,C 180,E1 4561.832,E2 4561.832} C_VEL
LIN {X 0,Y 526.817,Z 1017.821,A -85,B 0,C 180,E1 4565.491,E2 4565.491} C_VEL
LIN {X 0,Y 525.082,Z 1044.27,A -85,B 0,C 180,E1 4569.555,E2 4569.555} C_VEL
LIN {X 0,Y 524.084,Z 1064.72,A -85,B 0,C 180,E1 4573.641,E2 4573.641} C_VEL
LIN {X 0,Y 523.365,Z 1081.774,A -85,B 0,C 180,E1 4578.317,E2 4578.317} C_VEL
LIN {X 0,Y 523.193,Z 1091.918,A -85,B 0,C 180,E1 4582.518,E2 4582.518} C_VEL
LIN {X 0,Y 523.103,Z 1097.627,A -85,B 0,C 180,E1 4586.681,E2 4586.681} C_VEL
LIN {X 0,Y 523.066,Z 1099,A -85,B 0,C 180,E1 4590,E2 4590} C_VEL
LIN {X 0,Y 523.102,Z 1097.628,A -85,B 0,C 180,E1 4593.318,E2 4593.318} C_VEL
LIN {X 0,Y 523.256,Z 1091.918,A -85,B 0,C 180,E1 4597.481,E2 4597.481} C_VEL
LIN {X 0,Y 523.371,Z 1081.776,A -85,B 0,C 180,E1 4601.683,E2 4601.683} C_VEL
LIN {X 0,Y 523.907,Z 1066.494,A -85,B 0,C 180,E1 4605.934,E2 4605.934} C_VEL
LIN {X 0,Y 524.952,Z 1045.385,A -85,B 0,C 180,E1 4610.248,E2 4610.248} C_VEL
LIN {X 0,Y 526.699,Z 1019.261,A -85,B 0,C 180,E1 4614.312,E2 4614.312} C_VEL
LIN {X 0,Y 529.011,Z 989.214,A -85,B 0,C 180,E1 4617.945,E2 4617.945} C_VEL
LIN {X 0,Y 531.714,Z 955.258,A -85,B 0,C 180,E1 4621.141,E2 4621.141} C_VEL
LIN {X 0,Y 534.549,Z 917.908,A -85,B 0,C 180,E1 4623.818,E2 4623.818} C_VEL
LIN {X 0,Y 537.154,Z 878.525,A -85,B 0,C 180,E1 4625.879,E2 4625.879} C_VEL
LIN {X 0,Y 539.099,Z 836.903,A -85,B 0,C 180,E1 4627.333,E2 4627.333} C_VEL
LIN {X 0,Y 540.1,Z 779.3,A -85,B 0,C 180,E1 4628.421,E2 4628.421} C_VEL
LIN {X 0,Y 539.409,Z 770.495,A -85,B 0,C 180,E1 4628.626,E2 4628.626} C_VEL
LIN {X 0,Y 522.463,Z 738.654,A -85,B 0,C 180,E1 4630.657,E2 4630.657} C_VEL
LIN {X 0,Y 522.324,Z 737.44,A -85,B 0,C 180,E1 4630.835,E2 4630.835} C_VEL
LIN {X 0,Y 522.395,Z 737.44,A -85,B 0,C 180,E1 4636.431,E2 4636.431} C_VEL
LIN {X 0,Y 522.292,Z 737.44,A -85,B 0,C 180,E1 4642.5,E2 4642.5} C_VEL
LIN {X 0,Y 522.304,Z 737.44,A -85,B 0,C 180,E1 4648.547,E2 4648.547} C_VEL
LIN {X 0,Y 522.509,Z 737.44,A -85,B 0,C 180,E1 4654.236,E2 4654.236} C_VEL
LIN {X 0,Y 522.62,Z 737.44,A -85,B 0,C 180,E1 4659.655,E2 4659.655} C_VEL
LIN {X 0,Y 522.494,Z 737.44,A -85,B 0,C 180,E1 4664.88,E2 4664.88} C_VEL
LIN {X 0,Y 522.715,Z 737.44,A -85,B 0,C 180,E1 4669.989,E2 4669.989} C_VEL
LIN {X 0,Y 522.864,Z 737.44,A -85,B 0,C 180,E1 4675.013,E2 4675.013} C_VEL
LIN {X 0,Y 522.896,Z 737.44,A -85,B 0,C 180,E1 4679.996,E2 4679.996} C_VEL
LIN {X 0,Y 522.849,Z 737.44,A -85,B 0,C 180,E1 4684.979,E2 4684.979} C_VEL
LIN {X 0,Y 522.761,Z 737.44,A -85,B 0,C 180,E1 4690.04,E2 4690.04} C_VEL
LIN {X 0,Y 522.652,Z 737.44,A -85,B 0,C 180,E1 4695.106,E2 4695.106} C_VEL
LIN {X 0,Y 522.59,Z 737.44,A -85,B 0,C 180,E1 4700.337,E2 4700.337} C_VEL
LIN {X 0,Y 522.423,Z 737.44,A -85,B 0,C 180,E1 4706.054,E2 4706.054} C_VEL
LIN {X 0,Y 522.343,Z 737.44,A -85,B 0,C 180,E1 4711.44,E2 4711.44} C_VEL
LIN {X 0,Y 522.244,Z 737.44,A -85,B 0,C 180,E1 4717.493,E2 4717.493} C_VEL
LIN {X 0,Y 522.36,Z 737.44,A -85,B 0,C 180,E1 4723.565,E2 4723.565} C_VEL
LIN {X 0,Y 522.384,Z 737.44,A -85,B 0,C 180,E1 4728.886,E2 4728.886} C_VEL
LIN {X 0,Y 522.287,Z 737.44,A -85,B 0,C 180,E1 4734.567,E2 4734.567} C_VEL
LIN {X 0,Y 522.313,Z 737.44,A -85,B 0,C 180,E1 4740.541,E2 4740.541} C_VEL
LIN {X 0,Y 531.869,Z 765.302,A -85,B 0,C 180,E1 4742.235,E2 4742.235} C_VEL
LIN {X 0,Y 530.298,Z 802.406,A -85,B 0,C 180,E1 4743.893,E2 4743.893} C_VEL
LIN {X 0,Y 528.487,Z 834.792,A -85,B 0,C 180,E1 4746.019,E2 4746.019} C_VEL
LIN {X 0,Y 526.652,Z 865.113,A -85,B 0,C 180,E1 4748.743,E2 4748.743} C_VEL
LIN {X 0,Y 525.102,Z 892.349,A -85,B 0,C 180,E1 4752.048,E2 4752.048} C_VEL
LIN {X 0,Y 524.096,Z 913.987,A -85,B 0,C 180,E1 4755.615,E2 4755.615} C_VEL
LIN {X 0,Y 523.511,Z 930.706,A -85,B 0,C 180,E1 4759.458,E2 4759.458} C_VEL
LIN {X 0,Y 523.239,Z 941.869,A -85,B 0,C 180,E1 4763.354,E2 4763.354} C_VEL
LIN {X 0,Y 523.142,Z 947.214,A -85,B 0,C 180,E1 4766.682,E2 4766.682} C_VEL
LIN {X 0,Y 523.17,Z 948.997,A -85,B 0,C 180,E1 4770,E2 4770} C_VEL
